  MoveL 674 to (56.44, 271.47, 190) mm, rotated rx -180 ry 0 rz -78.51 deg; joints [53.74, -26.691, 117.686, 53.744, 89.412, 89.198, -1451.486]
  MoveL 675 to (54.33, 277.32, 200) mm, rotated rx -180 ry 0 rz -72.32 deg; joints [53.369, -26.663, 117.257, 53.371, 89.646, 89.524, -1457.679]
  MoveL 676 to (51.74, 282.68, 210) mm, rotated rx 180 ry 0 rz -66.33 deg; joints [53.002, -26.629, 116.82, 53.002, 89.885, 89.848, -1463.668]
  MoveL 677 to (48.8, 287.5, 220) mm, rotated rx -180 ry 0 rz -60.59 deg; joints [52.638, -26.588, 116.376, 52.638, 90.129, 90.169, -1469.406]
  MoveL 678 to (45.62, 291.76, 230) mm, rotated rx -180 ry 0 rz -55.15 deg; joints [52.278, -26.54, 115.924, 52.28, 90.377, 90.487, -1474.846]
  MoveL 679 to (42.34, 295.45, 240) mm, rotated rx -180 ry 0 rz -50.06 deg; joints [51.921, -26.485, 115.464, 51.926, 90.63, 90.804, -1479.941]
  MoveL 680 to (39.07, 298.58, 250) mm, rotated rx -180 ry 0 rz -45.36 deg; joints [51.568, -26.422, 114.996, 51.577, 90.886, 91.117, -1484.643]
  MoveL 681 to (35.92, 301.18, 260) mm, rotated rx -180 ry 0 rz -41.09 deg; joints [51.218, -26.352, 114.52, 51.232, 91.147, 91.428, -1488.905]
  MoveL 682 to (33, 303.28, 270) mm, rotated rx -180 ry 0 rz -37.32 deg; joints [50.872, -26.275, 114.036, 50.893, 91.413, 91.737, -1492.679]
  MoveL 683 to (30.4, 304.94, 280) mm, rotated rx -180 ry 0 rz -34.08 deg; joints [50.529, -26.192, 113.545, 50.559, 91.682, 92.044, -1495.919]
  MoveL 684 to (28.22, 306.19, 290) mm, rotated rx -180 ry 0 rz -31.42 deg; joints [50.189, -26.102, 113.046, 50.229, 91.956, 92.348, -1498.582]
  MoveL 685 to (-21.11, 309.47, 290) mm, rotated rx 180 ry 0 rz 23.11 deg; joints [50.189, -26.125, 113.059, 50.229, 91.963, 92.356, -1553.11]
  Set speed (60.0 mm/s)
  MoveL 686 to (-18.74, 310.33, 280) mm, rotated rx -180 ry 0 rz 20.42 deg; joints [50.529, -26.229, 113.565, 50.559, 91.693, 92.057, -1550.424]
  MoveL 687 to (-15.8, 311.23, 270) mm, rotated rx -180 ry 0 rz 17.14 deg; joints [50.872, -26.331, 114.066, 50.894, 91.429, 91.757, -1547.138]
  MoveL 688 to (-12.3, 312.09, 260) mm, rotated rx 180 ry 0 rz 13.29 deg; joints [51.218, -26.429, 114.561, 51.233, 91.17, 91.456, -1543.29]
  MoveL 689 to (-8.28, 312.8, 250) mm, rotated rx -180 ry 0 rz 8.92 deg; joints [51.568, -26.522, 115.049, 51.577, 90.915, 91.154, -1538.917]
  MoveL 690 to (-3.78, 313.26, 240) mm, rotated rx -180 ry 0 rz 4.06 deg; joints [51.921, -26.61, 115.531, 51.926, 90.666, 90.85, -1534.059]
  MoveL 691 to (1.16, 313.37, 230) mm, rotated rx -180 ry 0 rz -1.24 deg; joints [52.278, -26.692, 116.005, 52.28, 90.42, 90.543, -1528.756]
  MoveL 692 to (6.46, 313.03, 220) mm, rotated rx -180 ry 0 rz -6.95 deg; joints [52.638, -26.768, 116.472, 52.639, 90.18, 90.235, -1523.053]
  MoveL 693 to (12.04, 312.14, 210) mm, rotated rx -180 ry 0 rz -13.01 deg; joints [53.002, -26.836, 116.931, 53.002, 89.943, 89.925, -1516.995]
  MoveL 694 to (17.8, 310.63, 200) mm, rotated rx -180 ry 0 rz -19.37 deg; joints [53.369, -26.897, 117.381, 53.37, 89.711, 89.611, -1510.629]
  MoveL 695 to (23.62, 308.44, 190) mm, rotated rx -180 ry 0 rz -25.99 deg; joints [53.74, -26.949, 117.823, 53.743, 89.483, 89.295, -1504.006]
  MoveL 696 to (29.38, 305.54, 180) mm, rotated rx -180 ry 0 rz -32.82 deg; joints [54.114, -26.993, 118.257, 54.121, 89.259, 88.976, -1497.176]
  MoveL 697 to (34.94, 301.92, 170) mm, rotated rx 180 ry 0 rz -39.81 deg; joints [54.492, -27.029, 118.682, 54.503, 89.04, 88.654, -1490.188]
  MoveL 698 to (40.17, 297.58, 160) mm, rotated rx -180 ry 0 rz -46.91 deg; joints [54.874, -27.057, 119.098, 54.891, 88.825, 88.33, -1483.094]
  MoveL 699 to (44.94, 292.58, 150) mm, rotated rx -180 ry 0 rz -54.06 deg; joints [55.259, -27.076, 119.507, 55.283, 88.615, 88.003, -1475.941]
  MoveL 700 to (49.15, 286.99, 140) mm, rotated rx -180 ry 0 rz -61.23 deg; joints [55.647, -27.089, 119.907, 55.68, 88.41, 87.673, -1468.774]
  MoveL 701 to (52.68, 280.9, 130) mm, rotated rx -180 ry 0 rz -68.36 deg; joints [56.04, -27.095, 120.299, 56.081, 88.211, 87.342, -1461.638]
  MoveL 702 to (55.46, 274.42, 120) mm, rotated rx -180 ry 0 rz -75.43 deg; joints [56.436, -27.096, 120.685, 56.488, 88.017, 87.009, -1454.572]
  MoveL 703 to (57.44, 267.68, 110) mm, rotated rx -180 ry 0 rz -82.39 deg; joints [56.835, -27.093, 121.064, 56.898, 87.829, 86.674, -1447.613]
  MoveL 704 to (58.6, 260.81, 100) mm, rotated rx 180 ry 0 rz -89.21 deg; joints [57.239, -27.086, 121.436, 57.314, 87.647, 86.34, -1440.794]
  MoveL 705 to (58.95, 253.96, 90) mm, rotated rx -180 ry 0 rz -95.85 deg; joints [57.646, -27.076, 121.803, 57.734, 87.472, 86.004, -1434.147]
  MoveL 706 to (58.51, 247.24, 80) mm, rotated rx -180 ry 0 rz -102.3 deg; joints [58.056, -27.066, 122.165, 58.158, 87.304, 85.669, -1427.701]
  MoveL 707 to (57.35, 240.79, 70) mm, rotated rx 180 ry 0 rz -108.52 deg; joints [58.471, -27.054, 122.522, 58.587, 87.144, 85.335, -1421.482]
  MoveL 708 to (55.55, 234.7, 60) mm, rotated rx -180 ry 0 rz -114.48 deg; joints [58.889, -27.042, 122.874, 59.02, 86.99, 85.002, -1415.517]
  MoveL 709 to (53.21, 229.07, 50) mm, rotated rx -180 ry 0 rz -120.17 deg; joints [59.311, -27.031, 123.223, 59.458, 86.844, 84.67, -1409.83]
  MoveL 710 to (50.45, 223.94, 40) mm, rotated rx -180 ry 0 rz -125.55 deg; joints [59.736, -27.021, 123.567, 59.899, 86.706, 84.34, -1404.447]
  MoveL 711 to (47.39, 219.37, 30) mm, rotated rx -180 ry 0 rz -130.61 deg; joints [60.166, -27.012, 123.907, 60.345, 86.576, 84.012, -1399.391]
  MoveL 712 to (44.15, 215.37, 20) mm, rotated rx -180 ry 0 rz -135.31 deg; joints [60.599, -27.005, 124.244, 60.794, 86.453, 83.685, -1394.688]
  MoveL 713 to (40.85, 211.93, 10) mm, rotated rx -180 ry 0 rz -139.64 deg; joints [61.035, -26.999, 124.577, 61.248, 86.339, 83.361, -1390.363]
  MoveL 714 to (37.62, 209.05, 0) mm, rotated rx -180 ry 0 rz -143.56 deg; joints [61.476, -26.994, 124.905, 61.705, 86.232, 83.039, -1386.442]
  MoveL 715 to (-21.11, 309.47, 290) mm, rotated rx 180 ry 0 rz 23.11 deg; joints [50.189, -26.125, 113.059, 50.229, 91.963, 92.356, -1553.11]
  Set speed (60.0 mm/s)
  MoveL 716 to (-34.79, 325.15, 290) mm, rotated rx -180 ry 0 rz 28.1 deg; joints [50.189, -24.773, 112.315, 50.215, 91.574, 91.889, -1558.101]
  MoveL 717 to (37.62, 209.05, 0) mm, rotated rx -180 ry 0 rz -143.56 deg; joints [61.476, -26.994, 124.905, 61.705, 86.232, 83.039, -1386.442]
  Set speed (60.0 mm/s)
  MoveL 718 to (55.59, 198.58, 0) mm, rotated rx -180 ry 0 rz -137.85 deg; joints [61.476, -25.55, 124.114, 61.745, 85.922, 82.463, -1392.15]
  MoveL 719 to (37.62, 209.05, 0) mm, rotated rx -180 ry 0 rz -143.56 deg; joints [61.476, -26.994, 124.905, 61.705, 86.232, 83.039, -1386.442]
  Set speed (60.0 mm/s)
  MoveL 720 to (40.85, 211.93, 10) mm, rotated rx 180 ry 0 rz -139.64 deg; joints [61.035, -26.999, 124.577, 61.248, 86.339, 83.361, -1390.363]
  MoveL 721 to (44.15, 215.37, 20) mm, rotated rx -180 ry 0 rz -135.31 deg; joints [60.599, -27.005, 124.244, 60.794, 86.453, 83.685, -1394.688]
  MoveL 722 to (47.39, 219.37, 30) mm, rotated rx -180 ry 0 rz -130.61 deg; joints [60.166, -27.012, 123.907, 60.345, 86.576, 84.012, -1399.391]
  MoveL 723 to (50.45, 223.94, 40) mm, rotated rx -180 ry 0 rz -125.55 deg; joints [59.736, -27.021, 123.567, 59.899, 86.706, 84.34, -1404.447]
  MoveL 724 to (53.21, 229.07, 50) mm, rotated rx -180 ry 0 rz -120.17 deg; joints [59.311, -27.031, 123.223, 59.458, 86.844, 84.67, -1409.83]
  MoveL 725 to (55.55, 234.7, 60) mm, rotated rx -180 ry 0 rz -114.48 deg; joints [58.889, -27.042, 122.874, 59.02, 86.99, 85.002, -1415.517]
  MoveL 726 to (57.35, 240.79, 70) mm, rotated rx -180 ry 0 rz -108.52 deg; joints [58.471, -27.054, 122.522, 58.587, 87.144, 85.335, -1421.482]
  MoveL 727 to (58.51, 247.24, 80) mm, rotated rx 180 ry 0 rz -102.3 deg; joints [58.056, -27.066, 122.165, 58.158, 87.304, 85.669, -1427.701]
  MoveL 728 to (58.95, 253.96, 90) mm, rotated rx -180 ry 0 rz -95.85 deg; joints [57.646, -27.076, 121.803, 57.734, 87.472, 86.004, -1434.147]
  MoveL 729 to (58.6, 260.81, 100) mm, rotated rx -180 ry 0 rz -89.21 deg; joints [57.239, -27.086, 121.436, 57.314, 87.647, 86.34, -1440.794]
  MoveL 730 to (57.44, 267.68, 110) mm, rotated rx -180 ry 0 rz -82.39 deg; joints [56.835, -27.093, 121.064, 56.898, 87.829, 86.674, -1447.613]
  MoveL 731 to (55.46, 274.42, 120) mm, rotated rx -180 ry 0 rz -75.43 deg; joints [56.436, -27.096, 120.685, 56.488, 88.017, 87.009, -1454.572]
  MoveL 732 to (52.68, 280.9, 130) mm, rotated rx -180 ry 0 rz -68.36 deg; joints [56.04, -27.095, 120.299, 56.081, 88.211, 87.342, -1461.638]
  MoveL 733 to (49.15, 286.99, 140) mm, rotated rx 180 ry 0 rz -61.23 deg; joints [55.647, -27.089, 119.907, 55.68, 88.41, 87.673, -1468.774]
  MoveL 734 to (44.94, 292.58, 150) mm, rotated rx -180 ry 0 rz -54.06 deg; joints [55.259, -27.076, 119.507, 55.283, 88.615, 88.003, -1475.941]
  MoveL 735 to (40.17, 297.58, 160) mm, rotated rx -180 ry 0 rz -46.91 deg; joints [54.874, -27.057, 119.098, 54.891, 88.825, 88.33, -1483.094]
  MoveL 736 to (34.94, 301.92, 170) mm, rotated rx -180 ry 0 rz -39.81 deg; joints [54.492, -27.029, 118.682, 54.503, 89.04, 88.654, -1490.188]
  MoveL 737 to (29.38, 305.54, 180) mm, rotated rx -180 ry 0 rz -32.82 deg; joints [54.114, -26.993, 118.257, 54.121, 89.259, 88.976, -1497.176]
  MoveL 738 to (23.62, 308.44, 190) mm, rotated rx -180 ry 0 rz -25.99 deg; joints [53.74, -26.949, 117.823, 53.743, 89.483, 89.295, -1504.006]
  MoveL 739 to (17.8, 310.63, 200) mm, rotated rx -180 ry 0 rz -19.37 deg; joints [53.369, -26.897, 117.381, 53.37, 89.711, 89.611, -1510.629]
  MoveL 740 to (12.04, 312.14, 210) mm, rotated rx 180 ry 0 rz -13.01 deg; joints [53.002, -26.836, 116.931, 53.002, 89.943, 89.925, -1516.995]
  MoveL 741 to (6.46, 313.03, 220) mm, rotated rx 180 ry 0 rz -6.95 deg; joints [52.638, -26.768, 116.472, 52.639, 90.18, 90.235, -1523.053]
  MoveL 742 to (1.16, 313.37, 230) mm, rotated rx 180 ry 0 rz -1.24 deg; joints [52.278, -26.692, 116.005, 52.28, 90.42, 90.543, -1528.756]
  MoveL 743 to (-3.78, 313.26, 240) mm, rotated rx -180 ry 0 rz 4.06 deg; joints [51.921, -26.61, 115.531, 51.926, 90.666, 90.85, -1534.059]
  MoveL 744 to (-8.28, 312.8, 250) mm, rotated rx -180 ry 0 rz 8.92 deg; joints [51.568, -26.522, 115.049, 51.577, 90.915, 91.154, -1538.917]
  MoveL 745 to (-12.3, 312.09, 260) mm, rotated rx -180 ry 0 rz 13.29 deg; joints [51.218, -26.429, 114.561, 51.233, 91.17, 91.456, -1543.29]
  MoveL 746 to (-15.8, 311.23, 270) mm, rotated rx -180 ry 0 rz 17.14 deg; joints [50.872, -26.331, 114.066, 50.894, 91.429, 91.757, -1547.138]
  MoveL 747 to (-18.74, 310.33, 280) mm, rotated rx -180 ry 0 rz 20.42 deg; joints [50.529, -26.229, 113.565, 50.559, 91.693, 92.057, -1550.424]
  MoveL 748 to (-21.11, 309.47, 290) mm, rotated rx -180 ry 0 rz 23.11 deg; joints [50.189, -26.125, 113.059, 50.229, 91.963, 92.356, -1553.11]
  MoveL 749 to (-34.79, 325.15, 290) mm, rotated rx -180 ry 0 rz 28.1 deg; joints [50.189, -24.773, 112.315, 50.215, 91.574, 91.889, -1558.101]
  Set speed (60.0 mm/s)
  MoveL 750 to (-31.73, 326.57, 280) mm, rotated rx -180 ry 0 rz 25.49 deg; joints [50.529, -24.874, 112.821, 50.547, 91.305, 91.585, -1555.486]
  MoveL 751 to (-27.92, 328.13, 270) mm, rotated rx -180 ry 0 rz 22.29 deg; joints [50.872, -24.972, 113.321, 50.883, 91.042, 91.281, -1552.288]
  MoveL 752 to (-23.38, 329.69, 260) mm, rotated rx 180 ry 0 rz 18.54 deg; joints [51.218, -25.067, 113.816, 51.225, 90.784, 90.976, -1548.542]
  MoveL 753 to (-18.11, 331.13, 250) mm, rotated rx -180 ry 0 rz 14.29 deg; joints [51.568, -25.158, 114.304, 51.571, 90.531, 90.669, -1544.286]
  MoveL 754 to (-12.17, 332.29, 240) mm, rotated rx -180 ry 0 rz 9.56 deg; joints [51.921, -25.244, 114.785, 51.922, 90.283, 90.361, -1539.557]
  MoveL 755 to (-5.61, 333.04, 230) mm, rotated rx 180 ry 0 rz 4.39 deg; joints [52.278, -25.324, 115.26, 52.278, 90.04, 90.051, -1534.392]
  MoveL 756 to (1.49, 333.22, 220) mm, rotated rx -180 ry 0 rz -1.17 deg; joints [52.638, -25.399, 115.727, 52.639, 89.801, 89.739, -1528.834]
  MoveL 757 to (9.03, 332.72, 210) mm, rotated rx -180 ry 0 rz -7.08 deg; joints [53.002, -25.466, 116.186, 53.004, 89.567, 89.425, -1522.922]
  MoveL 758 to (16.88, 331.41, 200) mm, rotated rx -180 ry 0 rz -13.3 deg; joints [53.369, -25.526, 116.636, 53.374, 89.337, 89.109, -1516.702]
  MoveL 759 to (24.89, 329.2, 190) mm, rotated rx -180 ry 0 rz -19.78 deg; joints [53.74, -25.578, 117.079, 53.749, 89.112, 88.789, -1510.217]
  MoveL 760 to (32.91, 326.04, 180) mm, rotated rx -180 ry 0 rz -26.49 deg; joints [54.114, -25.621, 117.512, 54.129, 88.892, 88.468, -1503.513]
  MoveL 761 to (40.75, 321.89, 170) mm, rotated rx -180 ry 0 rz -33.36 deg; joints [54.492, -25.656, 117.937, 54.514, 88.675, 88.143, -1496.637]
  MoveL 762 to (48.24, 316.75, 160) mm, rotated rx -180 ry 0 rz -40.37 deg; joints [54.874, -25.683, 118.353, 54.903, 88.464, 87.816, -1489.635]
  MoveL 763 to (55.2, 310.67, 150) mm, rotated rx -180 ry 0 rz -47.45 deg; joints [55.259, -25.702, 118.761, 55.297, 88.257, 87.486, -1482.551]
  MoveL 764 to (61.48, 303.74, 140) mm, rotated rx 180 ry 0 rz -54.57 deg; joints [55.647, -25.713, 119.16, 55.696, 88.056, 87.153, -1475.431]
  MoveL 765 to (66.92, 296.06, 130) mm, rotated rx -180 ry 0 rz -61.68 deg; joints [56.04, -25.718, 119.551, 56.099, 87.86, 86.819, -1468.317]
  MoveL 766 to (71.41, 287.77, 120) mm, rotated rx -180 ry 0 rz -68.75 deg; joints [56.436, -25.716, 119.935, 56.507, 87.669, 86.483, -1461.249]
  MoveL 767 to (74.87, 279.04, 110) mm, rotated rx -180 ry 0 rz -75.73 deg; joints [56.835, -25.71, 120.312, 56.92, 87.485, 86.145, -1454.266]
  MoveL 768 to (77.24, 270.04, 100) mm, rotated rx -180 ry 0 rz -82.6 deg; joints [57.239, -25.699, 120.682, 57.337, 87.306, 85.807, -1447.404]
  MoveL 769 to (78.53, 260.95, 90) mm, rotated rx -180 ry 0 rz -89.3 deg; joints [57.646, -25.686, 121.046, 57.759, 87.135, 85.468, -1440.696]
  MoveL 770 to (78.77, 251.96, 80) mm, rotated rx 180 ry 0 rz -95.83 deg; joints [58.056, -25.67, 121.404, 58.185, 86.97, 85.13, -1434.174]
  MoveL 771 to (78, 243.23, 70) mm, rotated rx -180 ry 0 rz -102.13 deg; joints [58.471, -25.653, 121.758, 58.616, 86.812, 84.791, -1427.868]
  MoveL 772 to (76.35, 234.91, 60) mm, rotated rx -180 ry 0 rz -108.19 deg; joints [58.889, -25.636, 122.106, 59.051, 86.662, 84.454, -1421.808]
  MoveL 773 to (73.92, 227.12, 50) mm, rotated rx -180 ry 0 rz -113.98 deg; joints [59.311, -25.619, 122.451, 59.49, 86.519, 84.117, -1416.021]
  MoveL 774 to (70.87, 219.96, 40) mm, rotated rx 180 ry 0 rz -119.46 deg; joints [59.736, -25.602, 122.791, 59.933, 86.384, 83.783, -1410.535]
  MoveL 775 to (67.34, 213.5, 30) mm, rotated rx -180 ry 0 rz -124.62 deg; joints [60.166, -25.587, 123.128, 60.38, 86.257, 83.45, -1405.378]
  MoveL 776 to (63.51, 207.78, 20) mm, rotated rx -180 ry 0 rz -129.42 deg; joints [60.599, -25.573, 123.46, 60.831, 86.137, 83.118, -1400.576]
  MoveL 777 to (59.54, 202.81, 10) mm, rotated rx -180 ry 0 rz -133.84 deg; joints [61.035, -25.561, 123.789, 61.286, 86.026, 82.79, -1396.157]
  MoveL 778 to (55.59, 198.58, 0) mm, rotated rx -180 ry 0 rz -137.85 deg; joints [61.476, -25.55, 124.114, 61.745, 85.922, 82.463, -1392.15]
  MoveL 779 to (-34.79, 325.15, 290) mm, rotated rx 180 ry 0 rz 28.1 deg; joints [50.189, -24.773, 112.315, 50.215, 91.574, 91.889, -1558.101]
  Set speed (60.0 mm/s)
  MoveL 780 to (-30.72, 304.75, 290) mm, rotated rx -180 ry 0 rz 34.47 deg; joints [50.189, -26.092, 113.041, 50.229, 91.953, 92.345, -1564.467]
  MoveL 781 to (55.59, 198.58, 0) mm, rotated rx -180 ry 0 rz -137.85 deg; joints [61.476, -25.55, 124.114, 61.745, 85.922, 82.463, -1392.15]
  Set speed (60.0 mm/s)
  MoveL 782 to (45.21, 216.6, 0) mm, rotated rx 180 ry 0 rz -133.83 deg; joints [61.476, -27.044, 124.932, 61.704, 86.242, 83.059, -1396.169]
  MoveL 783 to (55.59, 198.58, 0) mm, rotated rx -180 ry 0 rz -137.85 deg; joints [61.476, -25.55, 124.114, 61.745, 85.922, 82.463, -1392.15]
  Set speed (60.0 mm/s)
  MoveL 784 to (59.54, 202.81, 10) mm, rotated rx -180 ry 0 rz -133.84 deg; joints [61.035, -25.561, 123.789, 61.286, 86.026, 82.79, -1396.157]
  MoveL 785 to (63.51, 207.78, 20) mm, rotated rx -180 ry 0 rz -129.42 deg; joints [60.599, -25.573, 123.46, 60.831, 86.137, 83.118, -1400.576]
  MoveL 786 to (67.34, 213.5, 30) mm, rotated rx -180 ry 0 rz -124.62 deg; joints [60.166, -25.587, 123.128, 60.38, 86.257, 83.45, -1405.378]
  MoveL 787 to (70.87, 219.96, 40) mm, rotated rx -180 ry 0 rz -119.46 deg; joints [59.736, -25.602, 122.791, 59.933, 86.384, 83.783, -1410.535]
  MoveL 788 to (73.92, 227.12, 50) mm, rotated rx -180 ry 0 rz -113.98 deg; joints [59.311, -25.619, 122.451, 59.49, 86.519, 84.117, -1416.021]
  MoveL 789 to (76.35, 234.91, 60) mm, rotated rx -180 ry 0 rz -108.19 deg; joints [58.889, -25.636, 122.106, 59.051, 86.662, 84.454, -1421.808]
  MoveL 790 to (78, 243.23, 70) mm, rotated rx -180 ry 0 rz -102.13 deg; joints [58.471, -25.653, 121.758, 58.616, 86.812, 84.791, -1427.868]
  MoveL 791 to (78.77, 251.96, 80) mm, rotated rx -180 ry 0 rz -95.83 deg; joints [58.056, -25.67, 121.404, 58.185, 86.97, 85.13, -1434.174]
  MoveL 792 to (78.53, 260.95, 90) mm, rotated rx -180 ry 0 rz -89.3 deg; joints [57.646, -25.686, 121.046, 57.759, 87.135, 85.468, -1440.696]
  MoveL 793 to (77.24, 270.04, 100) mm, rotated rx 180 ry 0 rz -82.6 deg; joints [57.239, -25.699, 120.682, 57.337, 87.306, 85.807, -1447.404]
  MoveL 794 to (74.87, 279.04, 110) mm, rotated rx -180 ry 0 rz -75.73 deg; joints [56.835, -25.71, 120.312, 56.92, 87.485, 86.145, -1454.266]
  MoveL 795 to (71.41, 287.77, 120) mm, rotated rx 180 ry 0 rz -68.75 deg; joints [56.436, -25.716, 119.935, 56.507, 87.669, 86.483, -1461.249]
  MoveL 796 to (66.92, 296.06, 130) mm, rotated rx -180 ry 0 rz -61.68 deg; joints [56.04, -25.718, 119.551, 56.099, 87.86, 86.819, -1468.317]
  MoveL 797 to (61.48, 303.74, 140) mm, rotated rx 180 ry 0 rz -54.57 deg; joints [55.647, -25.713, 119.16, 55.696, 88.056, 87.153, -1475.431]
  MoveL 798 to (55.2, 310.67, 150) mm, rotated rx -180 ry 0 rz -47.45 deg; joints [55.259, -25.702, 118.761, 55.297, 88.257, 87.486, -1482.551]
  MoveL 799 to (48.24, 316.75, 160) mm, rotated rx -180 ry 0 rz -40.37 deg; joints [54.874, -25.683, 118.353, 54.903, 88.464, 87.816, -1489.635]
  MoveL 800 to (40.75, 321.89, 170) mm, rotated rx -180 ry 0 rz -33.36 deg; joints [54.492, -25.656, 117.937, 54.514, 88.675, 88.143, -1496.637]
  MoveL 801 to (32.91, 326.04, 180) mm, rotated rx -180 ry 0 rz -26.49 deg; joints [54.114, -25.621, 117.512, 54.129, 88.892, 88.468, -1503.513]
  MoveL 802 to (24.89, 329.2, 190) mm, rotated rx -180 ry 0 rz -19.78 deg; joints [53.74, -25.578, 117.079, 53.749, 89.112, 88.789, -1510.217]
  MoveL 803 to (16.88, 331.41, 200) mm, rotated rx -180 ry 0 rz -13.3 deg; joints [53.369, -25.526, 116.636, 53.374, 89.337, 89.109, -1516.702]
  MoveL 804 to (9.03, 332.72, 210) mm, rotated rx -180 ry 0 rz -7.08 deg; joints [53.002, -25.466, 116.186, 53.004, 89.567, 89.425, -1522.922]
  MoveL 805 to (1.49, 333.22, 220) mm, rotated rx -180 ry 0 rz -1.17 deg; joints [52.638, -25.399, 115.727, 52.639, 89.801, 89.739, -1528.834]
  MoveL 806 to (-5.61, 333.04, 230) mm, rotated rx 180 ry 0 rz 4.39 deg; joints [52.278, -25.324, 115.26, 52.278, 90.04, 90.051, -1534.392]
  MoveL 807 to (-12.17, 332.29, 240) mm, rotated rx 180 ry 0 rz 9.56 deg; joints [51.921, -25.244, 114.785, 51.922, 90.283, 90.361, -1539.557]
  MoveL 808 to (-18.11, 331.13, 250) mm, rotated rx -180 ry 0 rz 14.29 deg; joints [51.568, -25.158, 114.304, 51.571, 90.531, 90.669, -1544.286]
  MoveL 809 to (-23.38, 329.69, 260) mm, rotated rx -180 ry 0 rz 18.54 deg; joints [51.218, -25.067, 113.816, 51.225, 90.784, 90.976, -1548.542]
  MoveL 810 to (-27.92, 328.13, 270) mm, rotated rx -180 ry 0 rz 22.29 deg; joints [50.872, -24.972, 113.321, 50.883, 91.042, 91.281, -1552.288]
  MoveL 811 to (-31.73, 326.57, 280) mm, rotated rx -180 ry 0 rz 25.49 deg; joints [50.529, -24.874, 112.821, 50.547, 91.305, 91.585, -1555.486]
  MoveL 812 to (-34.79, 325.15, 290) mm, rotated rx -180 ry 0 rz 28.1 deg; joints [50.189, -24.773, 112.315, 50.215, 91.574, 91.889, -1558.101]
  MoveL 813 to (-30.72, 304.75, 290) mm, rotated rx 180 ry 0 rz 34.47 deg; joints [50.189, -26.092, 113.041, 50.229, 91.953, 92.345, -1564.467]
  Set speed (60.0 mm/s)
  MoveL 814 to (-28.54, 306.02, 280) mm, rotated rx -180 ry 0 rz 31.81 deg; joints [50.529, -26.199, 113.549, 50.559, 91.684, 92.046, -1561.806]
  MoveL 815 to (-25.81, 307.44, 270) mm, rotated rx 180 ry 0 rz 28.55 deg; joints [50.872, -26.304, 114.052, 50.893, 91.421, 91.748, -1558.548]
  MoveL 816 to (-22.53, 308.91, 260) mm, rotated rx -180 ry 0 rz 24.73 deg; joints [51.218, -26.406, 114.549, 51.233, 91.163, 91.448, -1554.728]
  MoveL 817 to (-18.7, 310.34, 250) mm, rotated rx -180 ry 0 rz 20.38 deg; joints [51.568, -26.504, 115.04, 51.577, 90.91, 91.147, -1550.381]
  MoveL 818 to (-14.35, 311.61, 240) mm, rotated rx 180 ry 0 rz 15.54 deg; joints [51.921, -26.598, 115.525, 51.926, 90.662, 90.845, -1545.543]
  MoveL 819 to (-9.52, 312.61, 230) mm, rotated rx -180 ry 0 rz 10.25 deg; joints [52.278, -26.687, 116.002, 52.28, 90.419, 90.541, -1540.254]
  MoveL 820 to (-4.24, 313.23, 220) mm, rotated rx -180 ry 0 rz 4.55 deg; joints [52.638, -26.769, 116.473, 52.639, 90.18, 90.236, -1534.554]
  MoveL 821 to (1.41, 313.37, 210) mm, rotated rx -180 ry 0 rz -1.51 deg; joints [53.002, -26.845, 116.935, 53.002, 89.946, 89.928, -1528.487]
  MoveL 822 to (7.35, 312.92, 200) mm, rotated rx -180 ry 0 rz -7.9 deg; joints [53.369, -26.913, 117.39, 53.37, 89.716, 89.617, -1522.098]
  MoveL 823 to (13.47, 311.83, 190) mm, rotated rx -180 ry 0 rz -14.57 deg; joints [53.74, -26.974, 117.836, 53.743, 89.49, 89.304, -1515.435]
  MoveL 824 to (19.65, 310.01, 180) mm, rotated rx -180 ry 0 rz -21.45 deg; joints [54.114, -27.026, 118.274, 54.121, 89.268, 88.988, -1508.548]
  MoveL 825 to (25.78, 307.45, 170) mm, rotated rx -180 ry 0 rz -28.51 deg; joints [54.492, -27.069, 118.703, 54.503, 89.051, 88.67, -1501.489]
  MoveL 826 to (31.7, 304.13, 160) mm, rotated rx 180 ry 0 rz -35.69 deg; joints [54.874, -27.104, 119.123, 54.89, 88.838, 88.348, -1494.307]
  MoveL 827 to (37.3, 300.08, 150) mm, rotated rx -180 ry 0 rz -42.95 deg; joints [55.259, -27.13, 119.535, 55.282, 88.63, 88.023, -1487.054]
  MoveL 828 to (42.45, 295.34, 140) mm, rotated rx -180 ry 0 rz -50.22 deg; joints [55.647, -27.148, 119.938, 55.679, 88.426, 87.696, -1479.778]
  MoveL 829 to (47.02, 289.99, 130) mm, rotated rx -180 ry 0 rz -57.48 deg; joints [56.04, -27.16, 120.334, 56.08, 88.228, 87.367, -1472.524]
  MoveL 830 to (50.93, 284.12, 120) mm, rotated rx -180 ry 0 rz -64.66 deg; joints [56.436, -27.164, 120.721, 56.487, 88.034, 87.035, -1465.337]
  MoveL 831 to (54.1, 277.85, 110) mm, rotated rx -180 ry 0 rz -71.74 deg; joints [56.835, -27.164, 121.101, 56.897, 87.847, 86.702, -1458.256]
  MoveL 832 to (56.49, 271.3, 100) mm, rotated rx -180 ry 0 rz -78.68 deg; joints [57.239, -27.158, 121.475, 57.313, 87.666, 86.368, -1451.316]
  MoveL 833 to (58.06, 264.62, 90) mm, rotated rx -180 ry 0 rz -85.45 deg; joints [57.646, -27.15, 121.842, 57.733, 87.491, 86.033, -1444.553]
  MoveL 834 to (58.85, 257.94, 80) mm, rotated rx -180 ry 0 rz -92 deg; joints [58.056, -27.138, 122.204, 58.157, 87.322, 85.698, -1437.997]
  MoveL 835 to (58.87, 251.39, 70) mm, rotated rx -180 ry 0 rz -98.32 deg; joints [58.471, -27.125, 122.56, 58.586, 87.161, 85.364, -1431.675]
  MoveL 836 to (58.2, 245.07, 60) mm, rotated rx -180 ry 0 rz -104.38 deg; joints [58.889, -27.112, 122.912, 59.019, 87.007, 85.03, -1425.616]
  MoveL 837 to (56.92, 239.11, 50) mm, rotated rx -180 ry 0 rz -110.16 deg; joints [59.311, -27.098, 123.259, 59.456, 86.86, 84.697, -1419.845]
  MoveL 838 to (55.13, 233.57, 40) mm, rotated rx -180 ry 0 rz -115.61 deg; joints [59.736, -27.085, 123.601, 59.898, 86.721, 84.366, -1414.385]
  MoveL 839 to (52.95, 228.52, 30) mm, rotated rx 180 ry 0 rz -120.74 deg; joints [60.166, -27.073, 123.94, 60.343, 86.59, 84.036, -1409.263]
  MoveL 840 to (50.48, 223.99, 20) mm, rotated rx -180 ry 0 rz -125.5 deg; joints [60.599, -27.062, 124.274, 60.793, 86.466, 83.708, -1404.503]
  MoveL 841 to (47.86, 220.02, 10) mm, rotated rx 180 ry 0 rz -129.87 deg; joints [61.035, -27.052, 124.605, 61.247, 86.35, 83.383, -1400.13]
  MoveL 842 to (45.21, 216.6, 0) mm, rotated rx 180 ry 0 rz -133.83 deg; joints [61.476, -27.044, 124.932, 61.704, 86.242, 83.059, -1396.169]
  MoveL 843 to (-30.72, 304.75, 290) mm, rotated rx -180 ry 0 rz 34.47 deg; joints [50.189, -26.092, 113.041, 50.229, 91.953, 92.345, -1564.467]
  Set speed (60.0 mm/s)
  MoveL 844 to (-58.22, 263.67, 290) mm, rotated rx -180 ry 0 rz 86.39 deg; joints [50.189, -25.818, 112.893, 50.226, 91.873, 92.248, -1616.394]
  MoveL 845 to (45.21, 216.6, 0) mm, rotated rx -180 ry 0 rz -133.83 deg; joints [61.476, -27.044, 124.932, 61.704, 86.242, 83.059, -1756.169]
  Set speed (60.0 mm/s)
  MoveL 846 to (58.12, 264.32, 0) mm, rotated rx 180 ry 0 rz -85.75 deg; joints [61.476, -27.37, 125.106, 61.695, 86.315, 83.194, -1804.254]
  MoveL 847 to (45.21, 216.6, 0) mm, rotated rx -180 ry 0 rz -133.83 deg; joints [61.476, -27.044, 124.932, 61.704, 86.242, 83.059, -1756.169]
  Set speed (60.0 mm/s)
  MoveL 848 to (47.86, 220.02, 10) mm, rotated rx -180 ry 0 rz -129.87 deg; joints [61.035, -27.052, 124.605, 61.247, 86.35, 83.383, -1760.13]
  MoveL 849 to (50.48, 223.99, 20) mm, rotated rx -180 ry 0 rz -125.5 deg; joints [60.599, -27.062, 124.274, 60.793, 86.466, 83.708, -1764.503]
  MoveL 850 to (52.95, 228.52, 30) mm, rotated rx -180 ry 0 rz -120.74 deg; joints [60.166, -27.073, 123.94, 60.343, 86.59, 84.036, -1769.263]
  MoveL 851 to (55.13, 233.57, 40) mm, rotated rx 180 ry 0 rz -115.61 deg; joints [59.736, -27.085, 123.601, 59.898, 86.721, 84.366, -1774.385]
  MoveL 852 to (56.92, 239.11, 50) mm, rotated rx -180 ry 0 rz -110.16 deg; joints [59.311, -27.098, 123.259, 59.456, 86.86, 84.697, -1779.845]
  MoveL 853 to (58.2, 245.07, 60) mm, rotated rx -180 ry 0 rz -104.38 deg; joints [58.889, -27.112, 122.912, 59.019, 87.007, 85.03, -1785.616]
  MoveL 854 to (58.87, 251.39, 70) mm, rotated rx -180 ry 0 rz -98.32 deg; joints [58.471, -27.125, 122.56, 58.586, 87.161, 85.364, -1791.675]
  MoveL 855 to (58.85, 257.94, 80) mm, rotated rx 180 ry 0 rz -92 deg; joints [58.056, -27.138, 122.204, 58.157, 87.322, 85.698, -1797.997]
  MoveL 856 to (58.06, 264.62, 90) mm, rotated rx -180 ry 0 rz -85.45 deg; joints [57.646, -27.15, 121.842, 57.733, 87.491, 86.033, -1804.553]
  MoveL 857 to (56.49, 271.3, 100) mm, rotated rx -180 ry 0 rz -78.68 deg; joints [57.239, -27.158, 121.475, 57.313, 87.666, 86.368, -1811.316]
  MoveL 858 to (54.1, 277.85, 110) mm, rotated rx -180 ry 0 rz -71.74 deg; joints [56.835, -27.164, 121.101, 56.897, 87.847, 86.702, -1818.256]
  MoveL 859 to (50.93, 284.12, 120) mm, rotated rx -180 ry 0 rz -64.66 deg; joints [56.436, -27.164, 120.721, 56.487, 88.034, 87.035, -1825.337]
  MoveL 860 to (47.02, 289.99, 130) mm, rotated rx 180 ry 0 rz -57.48 deg; joints [56.04, -27.16, 120.334, 56.08, 88.228, 87.367, -1832.524]
  MoveL 861 to (42.45, 295.34, 140) mm, rotated rx -180 ry 0 rz -50.22 deg; joints [55.647, -27.148, 119.938, 55.679, 88.426, 87.696, -1839.778]
  MoveL 862 to (37.3, 300.08, 150) mm, rotated rx -180 ry 0 rz -42.95 deg; joints [55.259, -27.13, 119.535, 55.282, 88.63, 88.023, -1847.054]
  MoveL 863 to (31.7, 304.13, 160) mm, rotated rx -180 ry 0 rz -35.69 deg; joints [54.874, -27.104, 119.123, 54.89, 88.838, 88.348, -1854.307]
  MoveL 864 to (25.78, 307.45, 170) mm, rotated rx -180 ry 0 rz -28.51 deg; joints [54.492, -27.069, 118.703, 54.503, 89.051, 88.67, -1861.489]
  MoveL 865 to (19.65, 310.01, 180) mm, rotated rx 180 ry 0 rz -21.45 deg; joints [54.114, -27.026, 118.274, 54.121, 89.268, 88.988, -1868.548]
  MoveL 866 to (13.47, 311.83, 190) mm, rotated rx -180 ry 0 rz -14.57 deg; joints [53.74, -26.974, 117.836, 53.743, 89.49, 89.304, -1875.435]
  MoveL 867 to (7.35, 312.92, 200) mm, rotated rx -180 ry 0 rz -7.9 deg; joints [53.369, -26.913, 117.39, 53.37, 89.716, 89.617, -1882.098]
  MoveL 868 to (1.41, 313.37, 210) mm, rotated rx -180 ry 0 rz -1.51 deg; joints [53.002, -26.845, 116.935, 53.002, 89.946, 89.928, -1888.487]
  MoveL 869 to (-4.24, 313.23, 220) mm, rotated rx 180 ry 0 rz 4.55 deg; joints [52.638, -26.769, 116.473, 52.639, 90.18, 90.236, -1894.554]
  MoveL 870 to (-9.52, 312.61, 230) mm, rotated rx 180 ry 0 rz 10.25 deg; joints [52.278, -26.687, 116.002, 52.28, 90.419, 90.541, -1900.254]
  MoveL 871 to (-14.35, 311.61, 240) mm, rotated rx -180 ry 0 rz 15.54 deg; joints [51.921, -26.598, 115.525, 51.926, 90.662, 90.845, -1905.543]
  MoveL 872 to (-18.7, 310.34, 250) mm, rotated rx -180 ry 0 rz 20.38 deg; joints [51.568, -26.504, 115.04, 51.577, 90.91, 91.147, -1910.381]
  MoveL 873 to (-22.53, 308.91, 260) mm, rotated rx 180 ry 0 rz 24.73 deg; joints [51.218, -26.406, 114.549, 51.233, 91.163, 91.448, -1914.728]
  MoveL 874 to (-25.81, 307.44, 270) mm, rotated rx -180 ry 0 rz 28.55 deg; joints [50.872, -26.304, 114.052, 50.893, 91.421, 91.748, -1918.548]
  MoveL 875 to (-28.54, 306.02, 280) mm, rotated rx -180 ry 0 rz 31.81 deg; joints [50.529, -26.199, 113.549, 50.559, 91.684, 92.046, -1921.806]
  MoveL 876 to (-30.72, 304.75, 290) mm, rotated rx -180 ry 0 rz 34.47 deg; joints [50.189, -26.092, 113.041, 50.229, 91.953, 92.345, -1924.467]
  MoveL 877 to (-58.22, 263.67, 290) mm, rotated rx -180 ry 0 rz 86.39 deg; joints [50.189, -25.818, 112.893, 50.226, 91.873, 92.248, -1976.394]
  Set speed (60.0 mm/s)
  MoveL 878 to (-57.77, 266.15, 280) mm, rotated rx 180 ry 0 rz 83.92 deg; joints [50.529, -25.932, 113.405, 50.556, 91.606, 91.951, -1973.924]
  MoveL 879 to (-57.08, 269.15, 270) mm, rotated rx -180 ry 0 rz 80.89 deg; joints [50.872, -26.045, 113.912, 50.891, 91.346, 91.655, -1970.894]
  MoveL 880 to (-56.08, 272.6, 260) mm, rotated rx -180 ry 0 rz 77.33 deg; joints [51.218, -26.159, 114.416, 51.231, 91.092, 91.359, -1967.333]
  MoveL 881 to (-54.69, 276.44, 250) mm, rotated rx -180 ry 0 rz 73.27 deg; joints [51.568, -26.271, 114.915, 51.576, 90.843, 91.063, -1963.267]
  MoveL 882 to (-52.84, 280.57, 240) mm, rotated rx 180 ry 0 rz 68.72 deg; joints [51.921, -26.383, 115.409, 51.925, 90.601, 90.767, -1958.724]
  MoveL 883 to (-50.46, 284.91, 230) mm, rotated rx -180 ry 0 rz 63.73 deg; joints [52.278, -26.493, 115.899, 52.28, 90.364, 90.47, -1953.731]
  MoveL 884 to (-47.51, 289.33, 220) mm, rotated rx -180 ry 0 rz 58.32 deg; joints [52.638, -26.601, 116.383, 52.638, 90.132, 90.173, -1948.316]
  MoveL 885 to (-43.95, 293.72, 210) mm, rotated rx -180 ry 0 rz 52.51 deg; joints [53.002, -26.705, 116.861, 53.002, 89.906, 89.876, -1942.509]
  MoveL 886 to (-39.77, 297.95, 200) mm, rotated rx -180 ry 0 rz 46.34 deg; joints [53.369, -26.806, 117.333, 53.37, 89.686, 89.577, -1936.342]
  MoveL 887 to (-34.96, 301.9, 190) mm, rotated rx -180 ry 0 rz 39.85 deg; joints [53.74, -26.902, 117.798, 53.743, 89.47, 89.277, -1929.847]
  MoveL 888 to (-29.57, 305.43, 180) mm, rotated rx 180 ry 0 rz 33.06 deg; joints [54.114, -26.992, 118.256, 54.121, 89.259, 88.976, -1923.063]
  MoveL 889 to (-23.65, 308.43, 170) mm, rotated rx -180 ry 0 rz 26.03 deg; joints [54.492, -27.076, 118.707, 54.503, 89.053, 88.672, -1916.03]
  MoveL 890 to (-17.28, 310.79, 160) mm, rotated rx -180 ry 0 rz 18.79 deg; joints [54.874, -27.152, 119.149, 54.89, 88.851, 88.366, -1908.791]
  MoveL 891 to (-10.57, 312.43, 150) mm, rotated rx -180 ry 0 rz 11.39 deg; joints [55.259, -27.22, 119.583, 55.282, 88.654, 88.058, -1901.395]
  MoveL 892 to (-3.62, 313.27, 140) mm, rotated rx -180 ry 0 rz 3.89 deg; joints [55.647, -27.279, 120.008, 55.678, 88.461, 87.747, -1893.889]
  MoveL 893 to (3.42, 313.28, 130) mm, rotated rx -180 ry 0 rz -3.67 deg; joints [56.04, -27.329, 120.423, 56.078, 88.272, 87.433, -1886.327]
  MoveL 894 to (10.42, 312.46, 120) mm, rotated rx -180 ry 0 rz -11.24 deg; joints [56.436, -27.37, 120.83, 56.484, 88.088, 87.116, -1878.761]
  MoveL 895 to (17.25, 310.8, 110) mm, rotated rx -180 ry 0 rz -18.76 deg; joints [56.835, -27.402, 121.227, 56.894, 87.908, 86.796, -1871.243]
  MoveL 896 to (23.78, 308.38, 100) mm, rotated rx -180 ry 0 rz -26.18 deg; joints [57.239, -27.425, 121.616, 57.308, 87.733, 86.474, -1863.825]
  MoveL 897 to (29.89, 305.25, 90) mm, rotated rx -180 ry 0 rz -33.45 deg; joints [57.646, -27.44, 121.996, 57.728, 87.564, 86.149, -1856.554]
  MoveL 898 to (35.48, 301.51, 80) mm, rotated rx -180 ry 0 rz -40.52 deg; joints [58.056, -27.448, 122.368, 58.151, 87.399, 85.822, -1849.477]
  MoveL 899 to (40.49, 297.28, 70) mm, rotated rx -180 ry 0 rz -47.36 deg; joints [58.471, -27.45, 122.732, 58.579, 87.241, 85.494, -1842.636]
  MoveL 900 to (44.86, 292.68, 60) mm, rotated rx -180 ry 0 rz -53.93 deg; joints [58.889, -27.447, 123.089, 59.012, 87.088, 85.165, -1836.069]
  MoveL 901 to (48.58, 287.83, 50) mm, rotated rx -180 ry 0 rz -60.19 deg; joints [59.311, -27.439, 123.44, 59.449, 86.941, 84.835, -1829.813]
  MoveL 902 to (51.63, 282.88, 40) mm, rotated rx -180 ry 0 rz -66.1 deg; joints [59.736, -27.428, 123.784, 59.89, 86.802, 84.505, -1823.9]
  MoveL 903 to (54.06, 277.94, 30) mm, rotated rx -180 ry 0 rz -71.64 deg; joints [60.166, -27.415, 124.122, 60.335, 86.669, 84.175, -1818.36]
  MoveL 904 to (55.91, 273.13, 20) mm, rotated rx -180 ry 0 rz -76.78 deg; joints [60.599, -27.4, 124.455, 60.785, 86.543, 83.847, -1813.221]
  MoveL 905 to (57.23, 268.56, 10) mm, rotated rx -180 ry 0 rz -81.49 deg; joints [61.035, -27.385, 124.783, 61.238, 86.425, 83.519, -1808.51]
  MoveL 906 to (58.12, 264.32, 0) mm, rotated rx -180 ry 0 rz -85.75 deg; joints [61.476, -27.37, 125.106, 61.695, 86.315, 83.194, -1804.254]
  MoveL 907 to (-58.22, 263.67, 290) mm, rotated rx -180 ry 0 rz 86.39 deg; joints [50.189, -25.818, 112.893, 50.226, 91.873, 92.248, -1976.394]
  Set speed (60.0 mm/s)
  MoveL 908 to (-78.63, 259.66, 290) mm, rotated rx 180 ry 0 rz 90.25 deg; joints [50.189, -24.451, 112.133, 50.212, 91.484, 91.781, -1980.245]
  MoveL 909 to (58.12, 264.32, 0) mm, rotated rx 180 ry 0 rz -85.75 deg; joints [61.476, -27.37, 125.106, 61.695, 86.315, 83.194, -1804.254]
  Set speed (60.0 mm/s)
  MoveL 910 to (76.17, 274.65, 0) mm, rotated rx 180 ry 0 rz -79.11 deg; joints [61.476, -25.94, 124.331, 61.734, 86.004, 82.616, -1810.889]
  MoveL 911 to (58.12, 264.32, 0) mm, rotated rx -180 ry 0 rz -85.75 deg; joints [61.476, -27.37, 125.106, 61.695, 86.315, 83.194, -1804.254]
  Set speed (60.0 mm/s)
  MoveL 912 to (57.23, 268.56, 10) mm, rotated rx -180 ry 0 rz -81.49 deg; joints [61.035, -27.385, 124.783, 61.238, 86.425, 83.519, -1808.51]
  MoveL 913 to (55.91, 273.13, 20) mm, rotated rx -180 ry 0 rz -76.78 deg; joints [60.599, -27.4, 124.455, 60.785, 86.543, 83.847, -1813.221]
  MoveL 914 to (54.06, 277.94, 30) mm, rotated rx -180 ry 0 rz -71.64 deg; joints [60.166, -27.415, 124.122, 60.335, 86.669, 84.175, -1818.36]
  MoveL 915 to (51.63, 282.88, 40) mm, rotated rx -180 ry 0 rz -66.1 deg; joints [59.736, -27.428, 123.784, 59.89, 86.802, 84.505, -1823.9]
  MoveL 916 to (48.58, 287.83, 50) mm, rotated rx 180 ry 0 rz -60.19 deg; joints [59.311, -27.439, 123.44, 59.449, 86.941, 84.835, -1829.813]
  MoveL 917 to (44.86, 292.68, 60) mm, rotated rx 180 ry 0 rz -53.93 deg; joints [58.889, -27.447, 123.089, 59.012, 87.088, 85.165, -1836.069]
  MoveL 918 to (40.49, 297.28, 70) mm, rotated rx -180 ry 0 rz -47.36 deg; joints [58.471, -27.45, 122.732, 58.579, 87.241, 85.494, -1842.636]
  MoveL 919 to (35.48, 301.51, 80) mm, rotated rx -180 ry 0 rz -40.52 deg; joints [58.056, -27.448, 122.368, 58.151, 87.399, 85.822, -1849.477]
  MoveL 920 to (29.89, 305.25, 90) mm, rotated rx -180 ry 0 rz -33.45 deg; joints [57.646, -27.44, 121.996, 57.728, 87.564, 86.149, -1856.554]
  MoveL 921 to (23.78, 308.38, 100) mm, rotated rx -180 ry 0 rz -26.18 deg; joints [57.239, -27.425, 121.616, 57.308, 87.733, 86.474, -1863.825]
  MoveL 922 to (17.25, 310.8, 110) mm, rotated rx -180 ry 0 rz -18.76 deg; joints [56.835, -27.402, 121.227, 56.894, 87.908, 86.796, -1871.243]
  MoveL 923 to (10.42, 312.46, 120) mm, rotated rx -180 ry 0 rz -11.24 deg; joints [56.436, -27.37, 120.83, 56.484, 88.088, 87.116, -1878.761]
  MoveL 924 to (3.42, 313.28, 130) mm, rotated rx -180 ry 0 rz -3.67 deg; joints [56.04, -27.329, 120.423, 56.078, 88.272, 87.433, -1886.327]
  MoveL 925 to (-3.62, 313.27, 140) mm, rotated rx -180 ry 0 rz 3.89 deg; joints [55.647, -27.279, 120.008, 55.678, 88.461, 87.747, -1893.889]
  MoveL 926 to (-10.57, 312.43, 150) mm, rotated rx -180 ry 0 rz 11.39 deg; joints [55.259, -27.22, 119.583, 55.282, 88.654, 88.058, -1901.395]
  MoveL 927 to (-17.28, 310.79, 160) mm, rotated rx -180 ry 0 rz 18.79 deg; joints [54.874, -27.152, 119.149, 54.89, 88.851, 88.366, -1908.791]
  MoveL 928 to (-23.65, 308.43, 170) mm, rotated rx -180 ry 0 rz 26.03 deg; joints [54.492, -27.076, 118.707, 54.503, 89.053, 88.672, -1916.03]
  MoveL 929 to (-29.57, 305.43, 180) mm, rotated rx -180 ry 0 rz 33.06 deg; joints [54.114, -26.992, 118.256, 54.121, 89.259, 88.976, -1923.063]
  MoveL 930 to (-34.96, 301.9, 190) mm, rotated rx 180 ry 0 rz 39.85 deg; joints [53.74, -26.902, 117.798, 53.743, 89.47, 89.277, -1929.847]
  MoveL 931 to (-39.77, 297.95, 200) mm, rotated rx -180 ry 0 rz 46.34 deg; joints [53.369, -26.806, 117.333, 53.37, 89.686, 89.577, -1936.342]
  MoveL 932 to (-43.95, 293.72, 210) mm, rotated rx -180 ry 0 rz 52.51 deg; joints [53.002, -26.705, 116.861, 53.002, 89.906, 89.876, -1942.509]
  MoveL 933 to (-47.51, 289.33, 220) mm, rotated rx -180 ry 0 rz 58.32 deg; joints [52.638, -26.601, 116.383, 52.638, 90.132, 90.173, -1948.316]
  MoveL 934 to (-50.46, 284.91, 230) mm, rotated rx 180 ry 0 rz 63.73 deg; joints [52.278, -26.493, 115.899, 52.28, 90.364, 90.47, -1953.731]
  MoveL 935 to (-52.84, 280.57, 240) mm, rotated rx -180 ry 0 rz 68.72 deg; joints [51.921, -26.383, 115.409, 51.925, 90.601, 90.767, -1958.724]
  MoveL 936 to (-54.69, 276.44, 250) mm, rotated rx -180 ry 0 rz 73.27 deg; joints [51.568, -26.271, 114.915, 51.576, 90.843, 91.063, -1963.267]
  MoveL 937 to (-56.08, 272.6, 260) mm, rotated rx -180 ry 0 rz 77.33 deg; joints [51.218, -26.159, 114.416, 51.231, 91.092, 91.359, -1967.333]
  MoveL 938 to (-57.08, 269.15, 270) mm, rotated rx -180 ry 0 rz 80.89 deg; joints [50.872, -26.045, 113.912, 50.891, 91.346, 91.655, -1970.894]
  MoveL 939 to (-57.77, 266.15, 280) mm, rotated rx -180 ry 0 rz 83.92 deg; joints [50.529, -25.932, 113.405, 50.556, 91.606, 91.951, -1973.924]
  MoveL 940 to (-58.22, 263.67, 290) mm, rotated rx -180 ry 0 rz 86.39 deg; joints [50.189, -25.818, 112.893, 50.226, 91.873, 92.248, -1976.394]
  MoveL 941 to (-78.63, 259.66, 290) mm, rotated rx -180 ry 0 rz 90.25 deg; joints [50.189, -24.451, 112.133, 50.212, 91.484, 91.781, -1980.245]
  Set speed (60.0 mm/s)
  MoveL 942 to (-78.34, 263.02, 280) mm, rotated rx -180 ry 0 rz 87.79 deg; joints [50.529, -24.56, 112.644, 50.544, 91.218, 91.479, -1977.792]
  MoveL 943 to (-77.78, 267.1, 270) mm, rotated rx 180 ry 0 rz 84.79 deg; joints [50.872, -24.669, 113.15, 50.881, 90.958, 91.178, -1974.787]
  MoveL 944 to (-76.86, 271.82, 260) mm, rotated rx -180 ry 0 rz 81.26 deg; joints [51.218, -24.777, 113.653, 51.224, 90.704, 90.877, -1971.259]
  MoveL 945 to (-75.48, 277.1, 250) mm, rotated rx 180 ry 0 rz 77.24 deg; joints [51.568, -24.886, 114.151, 51.57, 90.456, 90.575, -1967.238]
  MoveL 946 to (-73.51, 282.82, 240) mm, rotated rx -180 ry 0 rz 72.75 deg; joints [51.921, -24.993, 114.645, 51.922, 90.215, 90.274, -1962.753]
  MoveL 947 to (-70.88, 288.88, 230) mm, rotated rx 180 ry 0 rz 67.83 deg; joints [52.278, -25.099, 115.134, 52.278, 89.979, 89.972, -1957.833]
  MoveL 948 to (-67.49, 295.12, 220) mm, rotated rx 180 ry 0 rz 62.51 deg; joints [52.638, -25.203, 115.617, 52.639, 89.748, 89.67, -1952.509]
  MoveL 949 to (-63.28, 301.4, 210) mm, rotated rx -180 ry 0 rz 56.81 deg; joints [53.002, -25.304, 116.095, 53.005, 89.524, 89.368, -1946.81]
  MoveL 950 to (-58.22, 307.54, 200) mm, rotated rx -180 ry 0 rz 50.77 deg; joints [53.369, -25.401, 116.567, 53.375, 89.304, 89.064, -1940.77]
  MoveL 951 to (-52.31, 313.38, 190) mm, rotated rx -180 ry 0 rz 44.42 deg; joints [53.74, -25.495, 117.033, 53.75, 89.09, 88.76, -1934.421]
  MoveL 952 to (-45.56, 318.73, 180) mm, rotated rx -180 ry 0 rz 37.8 deg; joints [54.114, -25.583, 117.491, 54.129, 88.882, 88.454, -1927.8]
  MoveL 953 to (-38.04, 323.45, 170) mm, rotated rx -180 ry 0 rz 30.95 deg; joints [54.492, -25.664, 117.942, 54.514, 88.678, 88.146, -1920.945]
  MoveL 954 to (-29.85, 327.37, 160) mm, rotated rx 180 ry 0 rz 23.9 deg; joints [54.874, -25.739, 118.384, 54.902, 88.478, 87.836, -1913.897]
  MoveL 955 to (-21.11, 330.36, 150) mm, rotated rx -180 ry 0 rz 16.7 deg; joints [55.259, -25.806, 118.819, 55.296, 88.284, 87.524, -1906.697]
  MoveL 956 to (-11.96, 332.32, 140) mm, rotated rx -180 ry 0 rz 9.39 deg; joints [55.647, -25.865, 119.244, 55.694, 88.094, 87.209, -1899.391]
  MoveL 957 to (-2.59, 333.2, 130) mm, rotated rx -180 ry 0 rz 2.03 deg; joints [56.04, -25.915, 119.66, 56.096, 87.909, 86.892, -1892.026]
  MoveL 958 to (6.83, 332.94, 120) mm, rotated rx -180 ry 0 rz -5.35 deg; joints [56.436, -25.956, 120.067, 56.504, 87.728, 86.572, -1884.647]
  MoveL 959 to (16.13, 331.57, 110) mm, rotated rx -180 ry 0 rz -12.7 deg; joints [56.835, -25.988, 120.465, 56.916, 87.552, 86.25, -1877.302]
  MoveL 960 to (25.11, 329.13, 100) mm, rotated rx -180 ry 0 rz -19.96 deg; joints [57.239, -26.011, 120.854, 57.332, 87.381, 85.925, -1870.039]
  MoveL 961 to (33.62, 325.71, 90) mm, rotated rx -180 ry 0 rz -27.1 deg; joints [57.646, -26.026, 121.234, 57.753, 87.216, 85.597, -1862.902]
  MoveL 962 to (41.52, 321.41, 80) mm, rotated rx -180 ry 0 rz -34.06 deg; joints [58.056, -26.034, 121.606, 58.178, 87.056, 85.268, -1855.936]
  MoveL 963 to (48.7, 316.39, 70) mm, rotated rx -180 ry 0 rz -40.82 deg; joints [58.471, -26.035, 121.969, 58.608, 86.901, 84.937, -1849.182]
  MoveL 964 to (55.08, 310.79, 60) mm, rotated rx 180 ry 0 rz -47.32 deg; joints [58.889, -26.031, 122.326, 59.042, 86.752, 84.605, -1842.679]
  MoveL 965 to (60.61, 304.79, 50) mm, rotated rx -180 ry 0 rz -53.53 deg; joints [59.311, -26.022, 122.675, 59.48, 86.61, 84.272, -1836.465]
  MoveL 966 to (65.29, 298.57, 40) mm, rotated rx -180 ry 0 rz -59.43 deg; joints [59.736, -26.009, 123.017, 59.923, 86.475, 83.94, -1830.575]
  MoveL 967 to (69.12, 292.29, 30) mm, rotated rx -180 ry 0 rz -64.96 deg; joints [60.166, -25.994, 123.353, 60.37, 86.346, 83.607, -1825.041]
  MoveL 968 to (72.16, 286.11, 20) mm, rotated rx 180 ry 0 rz -70.1 deg; joints [60.599, -25.977, 123.684, 60.821, 86.225, 83.275, -1819.895]
  MoveL 969 to (74.48, 280.19, 10) mm, rotated rx -180 ry 0 rz -74.83 deg; joints [61.035, -25.958, 124.01, 61.275, 86.111, 82.945, -1815.168]
  MoveL 970 to (76.17, 274.65, 0) mm, rotated rx 180 ry 0 rz -79.11 deg; joints [61.476, -25.94, 124.331, 61.734, 86.004, 82.616, -1810.889]
  MoveL 971 to (-78.63, 259.66, 290) mm, rotated rx 180 ry 0 rz 90.25 deg; joints [50.189, -24.451, 112.133, 50.212, 91.484, 91.781, -1980.245]
  Set speed (60.0 mm/s)
  MoveL 972 to (-58.93, 252.99, 290) mm, rotated rx 180 ry 0 rz 96.78 deg; joints [50.189, -25.75, 112.856, 50.225, 91.853, 92.224, -1986.784]
  MoveL 973 to (76.17, 274.65, 0) mm, rotated rx 180 ry 0 rz -79.11 deg; joints [61.476, -25.94, 124.331, 61.734, 86.004, 82.616, -1810.889]
  Set speed (60.0 mm/s)
  MoveL 974 to (55.37, 274.67, 0) mm, rotated rx -180 ry 0 rz -75.16 deg; joints [61.476, -27.444, 125.145, 61.693, 86.331, 83.225, -1814.838]
  MoveL 975 to (76.17, 274.65, 0) mm, rotated rx -180 ry 0 rz -79.11 deg; joints [61.476, -25.94, 124.331, 61.734, 86.004, 82.616, -1810.889]
  Set speed (60.0 mm/s)
  MoveL 976 to (74.48, 280.19, 10) mm, rotated rx -180 ry 0 rz -74.83 deg; joints [61.035, -25.958, 124.01, 61.275, 86.111, 82.945, -1815.168]
  MoveL 977 to (72.16, 286.11, 20) mm, rotated rx -180 ry 0 rz -70.1 deg; joints [60.599, -25.977, 123.684, 60.821, 86.225, 83.275, -1819.895]
  MoveL 978 to (69.12, 292.29, 30) mm, rotated rx -180 ry 0 rz -64.96 deg; joints [60.166, -25.994, 123.353, 60.37, 86.346, 83.607, -1825.041]
  MoveL 979 to (65.29, 298.57, 40) mm, rotated rx -180 ry 0 rz -59.43 deg; joints [59.736, -26.009, 123.017, 59.923, 86.475, 83.94, -1830.575]
  MoveL 980 to (60.61, 304.79, 50) mm, rotated rx -180 ry 0 rz -53.53 deg; joints [59.311, -26.022, 122.675, 59.48, 86.61, 84.272, -1836.465]
  MoveL 981 to (55.08, 310.79, 60) mm, rotated rx -180 ry 0 rz -47.32 deg; joints [58.889, -26.031, 122.326, 59.042, 86.752, 84.605, -1842.679]
  MoveL 982 to (48.7, 316.39, 70) mm, rotated rx -180 ry 0 rz -40.82 deg; joints [58.471, -26.035, 121.969, 58.608, 86.901, 84.937, -1849.182]
  MoveL 983 to (41.52, 321.41, 80) mm, rotated rx -180 ry 0 rz -34.06 deg; joints [58.056, -26.034, 121.606, 58.178, 87.056, 85.268, -1855.936]
  MoveL 984 to (33.62, 325.71, 90) mm, rotated rx -180 ry 0 rz -27.1 deg; joints [57.646, -26.026, 121.234, 57.753, 87.216, 85.597, -1862.902]
  MoveL 985 to (25.11, 329.13, 100) mm, rotated rx -180 ry 0 rz -19.96 deg; joints [57.239, -26.011, 120.854, 57.332, 87.381, 85.925, -1870.039]
  MoveL 986 to (16.13, 331.57, 110) mm, rotated rx -180 ry 0 rz -12.7 deg; joints [56.835, -25.988, 120.465, 56.916, 87.552, 86.25, -1877.302]
  MoveL 987 to (6.83, 332.94, 120) mm, rotated rx 180 ry 0 rz -5.35 deg; joints [56.436, -25.956, 120.067, 56.504, 87.728, 86.572, -1884.647]
  MoveL 988 to (-2.59, 333.2, 130) mm, rotated rx 180 ry 0 rz 2.03 deg; joints [56.04, -25.915, 119.66, 56.096, 87.909, 86.892, -1892.026]
  MoveL 989 to (-11.96, 332.32, 140) mm, rotated rx -180 ry 0 rz 9.39 deg; joints [55.647, -25.865, 119.244, 55.694, 88.094, 87.209, -1899.391]
  MoveL 990 to (-21.11, 330.36, 150) mm, rotated rx -180 ry 0 rz 16.7 deg; joints [55.259, -25.806, 118.819, 55.296, 88.284, 87.524, -1906.697]
  MoveL 991 to (-29.85, 327.37, 160) mm, rotated rx -180 ry 0 rz 23.9 deg; joints [54.874, -25.739, 118.384, 54.902, 88.478, 87.836, -1913.897]
  MoveL 992 to (-38.04, 323.45, 170) mm, rotated rx -180 ry 0 rz 30.95 deg; joints [54.492, -25.664, 117.942, 54.514, 88.678, 88.146, -1920.945]
  MoveL 993 to (-45.56, 318.73, 180) mm, rotated rx 180 ry 0 rz 37.8 deg; joints [54.114, -25.583, 117.491, 54.129, 88.882, 88.454, -1927.8]
  MoveL 994 to (-52.31, 313.38, 190) mm, rotated rx -180 ry 0 rz 44.42 deg; joints [53.74, -25.495, 117.033, 53.75, 89.09, 88.76, -1934.421]
  MoveL 995 to (-58.22, 307.54, 200) mm, rotated rx 180 ry 0 rz 50.77 deg; joints [53.369, -25.401, 116.567, 53.375, 89.304, 89.064, -1940.77]
  MoveL 996 to (-63.28, 301.4, 210) mm, rotated rx -180 ry 0 rz 56.81 deg; joints [53.002, -25.304, 116.095, 53.005, 89.524, 89.368, -1946.81]
  MoveL 997 to (-67.49, 295.12, 220) mm, rotated rx 180 ry 0 rz 62.51 deg; joints [52.638, -25.203, 115.617, 52.639, 89.748, 89.67, -1952.509]
  MoveL 998 to (-70.88, 288.88, 230) mm, rotated rx -180 ry 0 rz 67.83 deg; joints [52.278, -25.099, 115.134, 52.278, 89.979, 89.972, -1957.833]
  MoveL 999 to (-73.51, 282.82, 240) mm, rotated rx -180 ry 0 rz 72.75 deg; joints [51.921, -24.993, 114.645, 51.922, 90.215, 90.274, -1962.753]
  MoveL 1000 to (-75.48, 277.1, 250) mm, rotated rx -180 ry 0 rz 77.24 deg; joints [51.568, -24.886, 114.151, 51.57, 90.456, 90.575, -1967.238]
  MoveL 1001 to (-76.86, 271.82, 260) mm, rotated rx -180 ry 0 rz 81.26 deg; joints [51.218, -24.777, 113.653, 51.224, 90.704, 90.877, -1971.259]
  MoveL 1002 to (-77.78, 267.1, 270) mm, rotated rx -180 ry 0 rz 84.79 deg; joints [50.872, -24.669, 113.15, 50.881, 90.958, 91.178, -1974.787]
  MoveL 1003 to (-78.34, 263.02, 280) mm, rotated rx 180 ry 0 rz 87.79 deg; joints [50.529, -24.56, 112.644, 50.544, 91.218, 91.479, -1977.792]
  MoveL 1004 to (-78.63, 259.66, 290) mm, rotated rx -180 ry 0 rz 90.25 deg; joints [50.189, -24.451, 112.133, 50.212, 91.484, 91.781, -1980.245]
  MoveL 1005 to (-58.93, 252.99, 290) mm, rotated rx -180 ry 0 rz 96.78 deg; joints [50.189, -25.75, 112.856, 50.225, 91.853, 92.224, -1986.784]
  Set speed (60.0 mm/s)
  MoveL 1006 to (-58.94, 255.51, 280) mm, rotated rx -180 ry 0 rz 94.36 deg; joints [50.529, -25.864, 113.367, 50.555, 91.586, 91.927, -1984.356]
  MoveL 1007 to (-58.8, 258.59, 270) mm, rotated rx -180 ry 0 rz 91.38 deg; joints [50.872, -25.977, 113.875, 50.891, 91.326, 91.631, -1981.378]
  MoveL 1008 to (-58.44, 262.16, 260) mm, rotated rx -180 ry 0 rz 87.88 deg; joints [51.218, -26.09, 114.379, 51.231, 91.072, 91.334, -1977.879]
  MoveL 1009 to (-57.77, 266.19, 250) mm, rotated rx -180 ry 0 rz 83.88 deg; joints [51.568, -26.204, 114.878, 51.575, 90.824, 91.038, -1973.884]
  MoveL 1010 to (-56.69, 270.59, 240) mm, rotated rx 180 ry 0 rz 79.42 deg; joints [51.921, -26.316, 115.373, 51.925, 90.582, 90.742, -1969.42]
  MoveL 1011 to (-55.14, 275.28, 230) mm, rotated rx -180 ry 0 rz 74.51 deg; joints [52.278, -26.428, 115.864, 52.279, 90.345, 90.446, -1964.512]
  MoveL 1012 to (-53.04, 280.16, 220) mm, rotated rx -180 ry 0 rz 69.19 deg; joints [52.638, -26.538, 116.349, 52.638, 90.115, 90.15, -1959.189]
  MoveL 1013 to (-50.33, 285.12, 210) mm, rotated rx -180 ry 0 rz 63.48 deg; joints [53.002, -26.646, 116.829, 53.002, 89.89, 89.854, -1953.477]
  MoveL 1014 to (-46.98, 290.04, 200) mm, rotated rx -180 ry 0 rz 57.4 deg; joints [53.369, -26.751, 117.303, 53.37, 89.67, 89.557, -1947.405]
  MoveL 1015 to (-42.97, 294.79, 190) mm, rotated rx 180 ry 0 rz 51 deg; joints [53.74, -26.852, 117.772, 53.743, 89.456, 89.258, -1941.005]
  MoveL 1016 to (-38.31, 299.24, 180) mm, rotated rx -180 ry 0 rz 44.31 deg; joints [54.114, -26.948, 118.233, 54.121, 89.247, 88.959, -1934.31]
  MoveL 1017 to (-33.03, 303.26, 170) mm, rotated rx -180 ry 0 rz 37.36 deg; joints [54.492, -27.039, 118.687, 54.503, 89.043, 88.658, -1927.357]
  MoveL 1018 to (-27.19, 306.74, 160) mm, rotated rx -180 ry 0 rz 30.19 deg; joints [54.874, -27.123, 119.133, 54.89, 88.843, 88.355, -1920.187]
  MoveL 1019 to (-20.88, 309.56, 150) mm, rotated rx 180 ry 0 rz 22.84 deg; joints [55.259, -27.199, 119.572, 55.282, 88.648, 88.05, -1912.844]
  MoveL 1020 to (-14.2, 311.65, 140) mm, rotated rx -180 ry 0 rz 15.37 deg; joints [55.647, -27.267, 120.001, 55.678, 88.458, 87.742, -1905.374]
  MoveL 1021 to (-7.28, 312.93, 130) mm, rotated rx -180 ry 0 rz 7.83 deg; joints [56.04, -27.327, 120.422, 56.078, 88.271, 87.432, -1897.828]
  MoveL 1022 to (-0.24, 313.38, 120) mm, rotated rx 180 ry 0 rz 0.26 deg; joints [56.436, -27.377, 120.834, 56.484, 88.09, 87.119, -1890.258]
  MoveL 1023 to (6.77, 312.99, 110) mm, rotated rx -180 ry 0 rz -7.29 deg; joints [56.835, -27.418, 121.236, 56.894, 87.913, 86.803, -1882.715]
  MoveL 1024 to (13.63, 311.79, 100) mm, rotated rx 180 ry 0 rz -14.75 deg; joints [57.239, -27.451, 121.63, 57.308, 87.74, 86.484, -1875.252]
  MoveL 1025 to (20.21, 309.81, 90) mm, rotated rx -180 ry 0 rz -22.08 deg; joints [57.646, -27.474, 122.014, 57.727, 87.572, 86.163, -1867.921]
  MoveL 1026 to (26.38, 307.15, 80) mm, rotated rx -180 ry 0 rz -29.23 deg; joints [58.056, -27.49, 122.39, 58.151, 87.41, 85.839, -1860.769]
  MoveL 1027 to (32.08, 303.89, 70) mm, rotated rx -180 ry 0 rz -36.16 deg; joints [58.471, -27.499, 122.758, 58.579, 87.253, 85.514, -1853.843]
  MoveL 1028 to (37.21, 300.16, 60) mm, rotated rx -180 ry 0 rz -42.82 deg; joints [58.889, -27.502, 123.118, 59.011, 87.101, 85.187, -1847.185]
  MoveL 1029 to (41.73, 296.07, 50) mm, rotated rx -180 ry 0 rz -49.17 deg; joints [59.311, -27.499, 123.471, 59.448, 86.956, 84.859, -1840.833]
  MoveL 1030 to (45.64, 291.75, 40) mm, rotated rx -180 ry 0 rz -55.18 deg; joints [59.736, -27.493, 123.818, 59.888, 86.817, 84.531, -1834.824]
  MoveL 1031 to (48.92, 287.33, 30) mm, rotated rx 180 ry 0 rz -60.81 deg; joints [60.166, -27.483, 124.158, 60.334, 86.685, 84.203, -1829.19]
  MoveL 1032 to (51.6, 282.93, 20) mm, rotated rx -180 ry 0 rz -66.04 deg; joints [60.599, -27.471, 124.492, 60.783, 86.56, 83.876, -1823.962]
  MoveL 1033 to (53.73, 278.68, 10) mm, rotated rx -180 ry 0 rz -70.83 deg; joints [61.035, -27.458, 124.821, 61.236, 86.442, 83.55, -1819.169]
  MoveL 1034 to (55.37, 274.67, 0) mm, rotated rx 180 ry 0 rz -75.16 deg; joints [61.476, -27.444, 125.145, 61.693, 86.331, 83.225, -1814.838]
  MoveL 1035 to (-58.93, 252.99, 290) mm, rotated rx 180 ry 0 rz 96.78 deg; joints [50.189, -25.75, 112.856, 50.225, 91.853, 92.224, -1986.784]
  Set speed (60.0 mm/s)
  MoveL 1036 to (-37.11, 208.63, 290) mm, rotated rx 180 ry 0 rz 144.16 deg; joints [50.189, -25.479, 112.707, 50.222, 91.774, 92.13, -2034.156]
  MoveL 1037 to (55.37, 274.67, 0) mm, rotated rx -180 ry 0 rz -75.16 deg; joints [61.476, -27.444, 125.145, 61.693, 86.331, 83.225, -2174.838]
  Set speed (60.0 mm/s)
  MoveL 1038 to (20.49, 309.71, 0) mm, rotated rx -180 ry 0 rz -22.4 deg; joints [61.476, -27.706, 125.283, 61.686, 86.39, 83.334, -2227.595]
  MoveL 1039 to (55.37, 274.67, 0) mm, rotated rx -180 ry 0 rz -75.16 deg; joints [61.476, -27.444, 125.145, 61.693, 86.331, 83.225, -2174.838]
  Set speed (60.0 mm/s)
  MoveL 1040 to (53.73, 278.68, 10) mm, rotated rx -180 ry 0 rz -70.83 deg; joints [61.035, -27.458, 124.821, 61.236, 86.442, 83.55, -2179.169]
  MoveL 1041 to (51.6, 282.93, 20) mm, rotated rx 180 ry 0 rz -66.04 deg; joints [60.599, -27.471, 124.492, 60.783, 86.56, 83.876, -2183.962]
  MoveL 1042 to (48.92, 287.33, 30) mm, rotated rx -180 ry 0 rz -60.81 deg; joints [60.166, -27.483, 124.158, 60.334, 86.685, 84.203, -2189.19]
  MoveL 1043 to (45.64, 291.75, 40) mm, rotated rx -180 ry 0 rz -55.18 deg; joints [59.736, -27.493, 123.818, 59.888, 86.817, 84.531, -2194.824]
  MoveL 1044 to (41.73, 296.07, 50) mm, rotated rx -180 ry 0 rz -49.17 deg; joints [59.311, -27.499, 123.471, 59.448, 86.956, 84.859, -2200.833]
  MoveL 1045 to (37.21, 300.16, 60) mm, rotated rx -180 ry 0 rz -42.82 deg; joints [58.889, -27.502, 123.118, 59.011, 87.101, 85.187, -2207.185]
  MoveL 1046 to (32.08, 303.89, 70) mm, rotated rx -180 ry 0 rz -36.16 deg; joints [58.471, -27.499, 122.758, 58.579, 87.253, 85.514, -2213.843]
  MoveL 1047 to (26.38, 307.15, 80) mm, rotated rx 180 ry 0 rz -29.23 deg; joints [58.056, -27.49, 122.39, 58.151, 87.41, 85.839, -2220.769]
  MoveL 1048 to (20.21, 309.81, 90) mm, rotated rx -180 ry 0 rz -22.08 deg; joints [57.646, -27.474, 122.014, 57.727, 87.572, 86.163, -2227.921]
  MoveL 1049 to (13.63, 311.79, 100) mm, rotated rx -180 ry 0 rz -14.75 deg; joints [57.239, -27.451, 121.63, 57.308, 87.74, 86.484, -2235.252]
  MoveL 1050 to (6.77, 312.99, 110) mm, rotated rx -180 ry 0 rz -7.29 deg; joints [56.835, -27.418, 121.236, 56.894, 87.913, 86.803, -2242.715]
  MoveL 1051 to (-0.24, 313.38, 120) mm, rotated rx -180 ry 0 rz 0.26 deg; joints [56.436, -27.377, 120.834, 56.484, 88.09, 87.119, -2250.258]
  MoveL 1052 to (-7.28, 312.93, 130) mm, rotated rx -180 ry 0 rz 7.83 deg; joints [56.04, -27.327, 120.422, 56.078, 88.271, 87.432, -2257.828]
  MoveL 1053 to (-14.2, 311.65, 140) mm, rotated rx -180 ry 0 rz 15.37 deg; joints [55.647, -27.267, 120.001, 55.678, 88.458, 87.742, -2265.374]
  MoveL 1054 to (-20.88, 309.56, 150) mm, rotated rx -180 ry 0 rz 22.84 deg; joints [55.259, -27.199, 119.572, 55.282, 88.648, 88.05, -2272.844]
  MoveL 1055 to (-27.19, 306.74, 160) mm, rotated rx 180 ry 0 rz 30.19 deg; joints [54.874, -27.123, 119.133, 54.89, 88.843, 88.355, -2280.187]
  MoveL 1056 to (-33.03, 303.26, 170) mm, rotated rx -180 ry 0 rz 37.36 deg; joints [54.492, -27.039, 118.687, 54.503, 89.043, 88.658, -2287.357]
  MoveL 1057 to (-38.31, 299.24, 180) mm, rotated rx 180 ry 0 rz 44.31 deg; joints [54.114, -26.948, 118.233, 54.121, 89.247, 88.959, -2294.31]
  MoveL 1058 to (-42.97, 294.79, 190) mm, rotated rx -180 ry 0 rz 51 deg; joints [53.74, -26.852, 117.772, 53.743, 89.456, 89.258, -2301.005]
  MoveL 1059 to (-46.98, 290.04, 200) mm, rotated rx -180 ry 0 rz 57.4 deg; joints [53.369, -26.751, 117.303, 53.37, 89.67, 89.557, -2307.405]
  MoveL 1060 to (-50.33, 285.12, 210) mm, rotated rx 180 ry 0 rz 63.48 deg; joints [53.002, -26.646, 116.829, 53.002, 89.89, 89.854, -2313.477]
  MoveL 1061 to (-53.04, 280.16, 220) mm, rotated rx 180 ry 0 rz 69.19 deg; joints [52.638, -26.538, 116.349, 52.638, 90.115, 90.15, -2319.189]
  MoveL 1062 to (-55.14, 275.28, 230) mm, rotated rx 180 ry 0 rz 74.51 deg; joints [52.278, -26.428, 115.864, 52.279, 90.345, 90.446, -2324.512]
  MoveL 1063 to (-56.69, 270.59, 240) mm, rotated rx 180 ry 0 rz 79.42 deg; joints [51.921, -26.316, 115.373, 51.925, 90.582, 90.742, -2329.42]
  MoveL 1064 to (-57.77, 266.19, 250) mm, rotated rx 180 ry 0 rz 83.88 deg; joints [51.568, -26.204, 114.878, 51.575, 90.824, 91.038, -2333.884]
  MoveL 1065 to (-58.44, 262.16, 260) mm, rotated rx -180 ry 0 rz 87.88 deg; joints [51.218, -26.09, 114.379, 51.231, 91.072, 91.334, -2337.879]
  MoveL 1066 to (-58.8, 258.59, 270) mm, rotated rx -180 ry 0 rz 91.38 deg; joints [50.872, -25.977, 113.875, 50.891, 91.326, 91.631, -2341.378]
  MoveL 1067 to (-58.94, 255.51, 280) mm, rotated rx -180 ry 0 rz 94.36 deg; joints [50.529, -25.864, 113.367, 50.555, 91.586, 91.927, -2344.356]
  MoveL 1068 to (-58.93, 252.99, 290) mm, rotated rx 180 ry 0 rz 96.78 deg; joints [50.189, -25.75, 112.856, 50.225, 91.853, 92.224, -2346.784]
  MoveL 1069 to (-37.11, 208.63, 290) mm, rotated rx -180 ry 0 rz 144.16 deg; joints [50.189, -25.479, 112.707, 50.222, 91.774, 92.13, -2394.156]
  Set speed (60.0 mm/s)
  MoveL 1070 to (-39.03, 210.26, 280) mm, rotated rx 180 ry 0 rz 141.88 deg; joints [50.529, -25.585, 113.215, 50.553, 91.506, 91.83, -2391.877]
  MoveL 1071 to (-41.29, 212.35, 270) mm, rotated rx -180 ry 0 rz 139.09 deg; joints [50.872, -25.69, 113.719, 50.888, 91.244, 91.53, -2389.089]
  MoveL 1072 to (-43.78, 214.95, 260) mm, rotated rx -180 ry 0 rz 135.82 deg; joints [51.218, -25.795, 114.218, 51.229, 90.988, 91.23, -2385.82]
  MoveL 1073 to (-46.4, 218.08, 250) mm, rotated rx -180 ry 0 rz 132.1 deg; joints [51.568, -25.9, 114.713, 51.574, 90.738, 90.93, -2382.097]
  MoveL 1074 to (-49.06, 221.75, 240) mm, rotated rx -180 ry 0 rz 127.95 deg; joints [51.921, -26.005, 115.205, 51.924, 90.494, 90.63, -2377.947]
  MoveL 1075 to (-51.62, 225.97, 230) mm, rotated rx -180 ry 0 rz 123.4 deg; joints [52.278, -26.11, 115.692, 52.279, 90.256, 90.331, -2373.396]
  MoveL 1076 to (-53.98, 230.73, 220) mm, rotated rx -180 ry 0 rz 118.47 deg; joints [52.638, -26.216, 116.175, 52.638, 90.025, 90.032, -2368.469]
  MoveL 1077 to (-56, 236.01, 210) mm, rotated rx 180 ry 0 rz 113.19 deg; joints [53.002, -26.322, 116.655, 53.002, 89.8, 89.734, -2363.192]
  MoveL 1078 to (-57.57, 241.75, 200) mm, rotated rx 180 ry 0 rz 107.59 deg; joints [53.369, -26.429, 117.13, 53.371, 89.581, 89.437, -2357.589]
  MoveL 1079 to (-58.59, 247.88, 190) mm, rotated rx -180 ry 0 rz 101.68 deg; joints [53.74, -26.535, 117.602, 53.745, 89.369, 89.14, -2351.684]
  MoveL 1080 to (-58.95, 254.32, 180) mm, rotated rx -180 ry 0 rz 95.5 deg; joints [54.114, -26.641, 118.069, 54.123, 89.163, 88.843, -2345.504]
  MoveL 1081 to (-58.59, 260.95, 170) mm, rotated rx -180 ry 0 rz 89.07 deg; joints [54.492, -26.745, 118.531, 54.505, 88.963, 88.547, -2339.073]
  MoveL 1082 to (-57.45, 267.65, 160) mm, rotated rx -180 ry 0 rz 82.42 deg; joints [54.874, -26.848, 118.987, 54.892, 88.769, 88.25, -2332.419]
  MoveL 1083 to (-55.51, 274.28, 150) mm, rotated rx -180 ry 0 rz 75.57 deg; joints [55.259, -26.948, 119.438, 55.284, 88.581, 87.953, -2325.573]
  MoveL 1084 to (-52.77, 280.72, 140) mm, rotated rx -180 ry 0 rz 68.57 deg; joints [55.647, -27.045, 119.883, 55.68, 88.399, 87.656, -2318.565]
  MoveL 1085 to (-49.26, 286.82, 130) mm, rotated rx -180 ry 0 rz 61.43 deg; joints [56.04, -27.137, 120.322, 56.081, 88.222, 87.358, -2311.431]
  MoveL 1086 to (-45.04, 292.47, 120) mm, rotated rx -180 ry 0 rz 54.21 deg; joints [56.436, -27.224, 120.753, 56.486, 88.05, 87.058, -2304.209]
  MoveL 1087 to (-40.19, 297.56, 110) mm, rotated rx -180 ry 0 rz 46.94 deg; joints [56.835, -27.304, 121.176, 56.895, 87.883, 86.758, -2296.94]
  MoveL 1088 to (-34.83, 302, 100) mm, rotated rx 180 ry 0 rz 39.67 deg; joints [57.239, -27.378, 121.591, 57.309, 87.721, 86.455, -2289.668]
  MoveL 1089 to (-29.06, 305.72, 90) mm, rotated rx -180 ry 0 rz 32.44 deg; joints [57.646, -27.444, 121.998, 57.728, 87.565, 86.15, -2282.441]
  MoveL 1090 to (-23.03, 308.7, 80) mm, rotated rx -180 ry 0 rz 25.31 deg; joints [58.056, -27.502, 122.396, 58.15, 87.413, 85.844, -2275.308]
  MoveL 1091 to (-16.86, 310.92, 70) mm, rotated rx 180 ry 0 rz 18.32 deg; joints [58.471, -27.552, 122.786, 58.577, 87.266, 85.535, -2268.32]
  MoveL 1092 to (-10.69, 312.41, 60) mm, rotated rx -180 ry 0 rz 11.53 deg; joints [58.889, -27.594, 123.167, 59.009, 87.124, 85.224, -2261.529]
  MoveL 1093 to (-4.64, 313.2, 50) mm, rotated rx 180 ry 0 rz 4.98 deg; joints [59.311, -27.628, 123.539, 59.445, 86.987, 84.912, -2254.983]
  MoveL 1094 to (1.18, 313.37, 40) mm, rotated rx -180 ry 0 rz -1.27 deg; joints [59.736, -27.655, 123.903, 59.885, 86.856, 84.598, -2248.733]
  MoveL 1095 to (6.67, 313.01, 30) mm, rotated rx -180 ry 0 rz -7.17 deg; joints [60.166, -27.676, 124.259, 60.329, 86.73, 84.283, -2242.826]
  MoveL 1096 to (11.76, 312.2, 20) mm, rotated rx -180 ry 0 rz -12.69 deg; joints [60.599, -27.69, 124.608, 60.777, 86.61, 83.967, -2237.306]
  MoveL 1097 to (16.38, 311.06, 10) mm, rotated rx -180 ry 0 rz -17.78 deg; joints [61.035, -27.7, 124.949, 61.23, 86.497, 83.65, -2232.216]
  MoveL 1098 to (20.49, 309.71, 0) mm, rotated rx -180 ry 0 rz -22.4 deg; joints [61.476, -27.706, 125.283, 61.686, 86.39, 83.334, -2227.595]
  MoveL 1099 to (-37.11, 208.63, 290) mm, rotated rx -180 ry 0 rz 144.16 deg; joints [50.189, -25.479, 112.707, 50.222, 91.774, 92.13, -2394.156]
  Set speed (60.0 mm/s)
  MoveL 1100 to (-43.85, 188.95, 290) mm, rotated rx -180 ry 0 rz 148.32 deg; joints [50.189, -24.124, 111.947, 50.209, 91.394, 91.673, -2398.321]
  MoveL 1101 to (20.49, 309.71, 0) mm, rotated rx -180 ry 0 rz -22.4 deg; joints [61.476, -27.706, 125.283, 61.686, 86.39, 83.334, -2227.595]
  Set speed (60.0 mm/s)
  MoveL 1102 to (20.57, 330.51, 0) mm, rotated rx -180 ry 0 rz -16.27 deg; joints [61.476, -26.245, 124.499, 61.726, 86.069, 82.736, -2233.733]
  MoveL 1103 to (20.49, 309.71, 0) mm, rotated rx -180 ry 0 rz -22.4 deg; joints [61.476, -27.706, 125.283, 61.686, 86.39, 83.334, -2227.595]
  Set speed (60.0 mm/s)
  MoveL 1104 to (16.38, 311.06, 10) mm, rotated rx -180 ry 0 rz -17.78 deg; joints [61.035, -27.7, 124.949, 61.23, 86.497, 83.65, -2232.216]
  MoveL 1105 to (11.76, 312.2, 20) mm, rotated rx -180 ry 0 rz -12.69 deg; joints [60.599, -27.69, 124.608, 60.777, 86.61, 83.967, -2237.306]
  MoveL 1106 to (6.67, 313.01, 30) mm, rotated rx -180 ry 0 rz -7.17 deg; joints [60.166, -27.676, 124.259, 60.329, 86.73, 84.283, -2242.826]
  MoveL 1107 to (1.18, 313.37, 40) mm, rotated rx -180 ry 0 rz -1.27 deg; joints [59.736, -27.655, 123.903, 59.885, 86.856, 84.598, -2248.733]
  MoveL 1108 to (-4.64, 313.2, 50) mm, rotated rx 180 ry 0 rz 4.98 deg; joints [59.311, -27.628, 123.539, 59.445, 86.987, 84.912, -2254.983]
  MoveL 1109 to (-10.69, 312.41, 60) mm, rotated rx -180 ry 0 rz 11.53 deg; joints [58.889, -27.594, 123.167, 59.009, 87.124, 85.224, -2261.529]
  MoveL 1110 to (-16.86, 310.92, 70) mm, rotated rx 180 ry 0 rz 18.32 deg; joints [58.471, -27.552, 122.786, 58.577, 87.266, 85.535, -2268.32]
  MoveL 1111 to (-23.03, 308.7, 80) mm, rotated rx -180 ry 0 rz 25.31 deg; joints [58.056, -27.502, 122.396, 58.15, 87.413, 85.844, -2275.308]
  MoveL 1112 to (-29.06, 305.72, 90) mm, rotated rx -180 ry 0 rz 32.44 deg; joints [57.646, -27.444, 121.998, 57.728, 87.565, 86.15, -2282.441]
  MoveL 1113 to (-34.83, 302, 100) mm, rotated rx -180 ry 0 rz 39.67 deg; joints [57.239, -27.378, 121.591, 57.309, 87.721, 86.455, -2289.668]
  MoveL 1114 to (-40.19, 297.56, 110) mm, rotated rx -180 ry 0 rz 46.94 deg; joints [56.835, -27.304, 121.176, 56.895, 87.883, 86.758, -2296.94]
  MoveL 1115 to (-45.04, 292.47, 120) mm, rotated rx -180 ry 0 rz 54.21 deg; joints [56.436, -27.224, 120.753, 56.486, 88.05, 87.058, -2304.209]
  MoveL 1116 to (-49.26, 286.82, 130) mm, rotated rx -180 ry 0 rz 61.43 deg; joints [56.04, -27.137, 120.322, 56.081, 88.222, 87.358, -2311.431]
  MoveL 1117 to (-52.77, 280.72, 140) mm, rotated rx -180 ry 0 rz 68.57 deg; joints [55.647, -27.045, 119.883, 55.68, 88.399, 87.656, -2318.565]
  MoveL 1118 to (-55.51, 274.28, 150) mm, rotated rx 180 ry 0 rz 75.57 deg; joints [55.259, -26.948, 119.438, 55.284, 88.581, 87.953, -2325.573]
  MoveL 1119 to (-57.45, 267.65, 160) mm, rotated rx 180 ry 0 rz 82.42 deg; joints [54.874, -26.848, 118.987, 54.892, 88.769, 88.25, -2332.419]
  MoveL 1120 to (-58.59, 260.95, 170) mm, rotated rx -180 ry 0 rz 89.07 deg; joints [54.492, -26.745, 118.531, 54.505, 88.963, 88.547, -2339.073]
  MoveL 1121 to (-58.95, 254.32, 180) mm, rotated rx 180 ry 0 rz 95.5 deg; joints [54.114, -26.641, 118.069, 54.123, 89.163, 88.843, -2345.504]
  MoveL 1122 to (-58.59, 247.88, 190) mm, rotated rx 180 ry 0 rz 101.68 deg; joints [53.74, -26.535, 117.602, 53.745, 89.369, 89.14, -2351.684]
  MoveL 1123 to (-57.57, 241.75, 200) mm, rotated rx -180 ry 0 rz 107.59 deg; joints [53.369, -26.429, 117.13, 53.371, 89.581, 89.437, -2357.589]
  MoveL 1124 to (-56, 236.01, 210) mm, rotated rx -180 ry 0 rz 113.19 deg; joints [53.002, -26.322, 116.655, 53.002, 89.8, 89.734, -2363.192]
  MoveL 1125 to (-53.98, 230.73, 220) mm, rotated rx -180 ry 0 rz 118.47 deg; joints [52.638, -26.216, 116.175, 52.638, 90.025, 90.032, -2368.469]
  MoveL 1126 to (-51.62, 225.97, 230) mm, rotated rx -180 ry 0 rz 123.4 deg; joints [52.278, -26.11, 115.692, 52.279, 90.256, 90.331, -2373.396]
  MoveL 1127 to (-49.06, 221.75, 240) mm, rotated rx -180 ry 0 rz 127.95 deg; joints [51.921, -26.005, 115.205, 51.924, 90.494, 90.63, -2377.947]
  MoveL 1128 to (-46.4, 218.08, 250) mm, rotated rx -180 ry 0 rz 132.1 deg; joints [51.568, -25.9, 114.713, 51.574, 90.738, 90.93, -2382.097]
  MoveL 1129 to (-43.78, 214.95, 260) mm, rotated rx -180 ry 0 rz 135.82 deg; joints [51.218, -25.795, 114.218, 51.229, 90.988, 91.23, -2385.82]
  MoveL 1130 to (-41.29, 212.35, 270) mm, rotated rx -180 ry 0 rz 139.09 deg; joints [50.872, -25.69, 113.719, 50.888, 91.244, 91.53, -2389.089]
  MoveL 1131 to (-39.03, 210.26, 280) mm, rotated rx -180 ry 0 rz 141.88 deg; joints [50.529, -25.585, 113.215, 50.553, 91.506, 91.83, -2391.877]
  MoveL 1132 to (-37.11, 208.63, 290) mm, rotated rx -180 ry 0 rz 144.16 deg; joints [50.189, -25.479, 112.707, 50.222, 91.774, 92.13, -2394.156]
  MoveL 1133 to (-43.85, 188.95, 290) mm, rotated rx 180 ry 0 rz 148.32 deg; joints [50.189, -24.124, 111.947, 50.209, 91.394, 91.673, -2398.321]
  Set speed (60.0 mm/s)
  MoveL 1134 to (-46.6, 190.89, 280) mm, rotated rx 180 ry 0 rz 146.01 deg; joints [50.529, -24.224, 112.453, 50.542, 91.126, 91.368, -2396.008]
  MoveL 1135 to (-49.86, 193.4, 270) mm, rotated rx -180 ry 0 rz 143.18 deg; joints [50.872, -24.324, 112.955, 50.88, 90.864, 91.062, -2393.179]
  MoveL 1136 to (-53.49, 196.56, 260) mm, rotated rx 180 ry 0 rz 139.86 deg; joints [51.218, -24.423, 113.452, 51.222, 90.608, 90.757, -2389.865]
  MoveL 1137 to (-57.36, 200.4, 250) mm, rotated rx -180 ry 0 rz 136.1 deg; joints [51.568, -24.521, 113.945, 51.569, 90.358, 90.451, -2386.095]
  MoveL 1138 to (-61.34, 204.96, 240) mm, rotated rx -180 ry 0 rz 131.9 deg; joints [51.921, -24.62, 114.435, 51.921, 90.115, 90.146, -2381.899]
  MoveL 1139 to (-65.27, 210.27, 230) mm, rotated rx -180 ry 0 rz 127.3 deg; joints [52.278, -24.719, 114.92, 52.278, 89.877, 89.841, -2377.303]
  MoveL 1140 to (-68.98, 216.33, 220) mm, rotated rx -180 ry 0 rz 122.34 deg; joints [52.638, -24.819, 115.402, 52.64, 89.646, 89.537, -2372.338]
  MoveL 1141 to (-72.31, 223.11, 210) mm, rotated rx -180 ry 0 rz 117.03 deg; joints [53.002, -24.919, 115.879, 53.006, 89.422, 89.233, -2367.029]
  MoveL 1142 to (-75.1, 230.56, 200) mm, rotated rx -180 ry 0 rz 111.4 deg; joints [53.369, -25.019, 116.353, 53.377, 89.204, 88.929, -2361.404]
  MoveL 1143 to (-77.2, 238.6, 190) mm, rotated rx -180 ry 0 rz 105.49 deg; joints [53.74, -25.12, 116.823, 53.752, 88.993, 88.626, -2355.49]
  MoveL 1144 to (-78.47, 247.13, 180) mm, rotated rx -180 ry 0 rz 99.32 deg; joints [54.114, -25.22, 117.289, 54.132, 88.788, 88.324, -2349.316]
  MoveL 1145 to (-78.79, 256, 170) mm, rotated rx -180 ry 0 rz 92.91 deg; joints [54.492, -25.32, 117.75, 54.517, 88.589, 88.021, -2342.909]
  MoveL 1146 to (-78.09, 265.05, 160) mm, rotated rx -180 ry 0 rz 86.3 deg; joints [54.874, -25.418, 118.206, 54.906, 88.396, 87.719, -2336.299]
  MoveL 1147 to (-76.31, 274.12, 150) mm, rotated rx -180 ry 0 rz 79.52 deg; joints [55.259, -25.513, 118.656, 55.299, 88.21, 87.417, -2329.517]
  MoveL 1148 to (-73.44, 283.02, 140) mm, rotated rx -180 ry 0 rz 72.6 deg; joints [55.647, -25.606, 119.1, 55.697, 88.029, 87.114, -2322.596]
  MoveL 1149 to (-69.5, 291.57, 130) mm, rotated rx -180 ry 0 rz 65.57 deg; joints [56.04, -25.694, 119.538, 56.099, 87.854, 86.81, -2315.57]
  MoveL 1150 to (-64.57, 299.61, 120) mm, rotated rx 180 ry 0 rz 58.48 deg; joints [56.436, -25.778, 119.969, 56.506, 87.684, 86.506, -2308.477]
  MoveL 1151 to (-58.74, 306.97, 110) mm, rotated rx -180 ry 0 rz 51.35 deg; joints [56.835, -25.856, 120.392, 56.918, 87.52, 86.2, -2301.355]
  MoveL 1152 to (-52.14, 313.53, 100) mm, rotated rx -180 ry 0 rz 44.25 deg; joints [57.239, -25.927, 120.808, 57.333, 87.361, 85.893, -2294.246]
  MoveL 1153 to (-44.91, 319.19, 90) mm, rotated rx -180 ry 0 rz 37.19 deg; joints [57.646, -25.991, 121.215, 57.753, 87.207, 85.584, -2287.194]
  MoveL 1154 to (-37.24, 323.88, 80) mm, rotated rx 180 ry 0 rz 30.24 deg; joints [58.056, -26.048, 121.613, 58.178, 87.059, 85.273, -2280.242]
  MoveL 1155 to (-29.3, 327.59, 70) mm, rotated rx -180 ry 0 rz 23.44 deg; joints [58.471, -26.097, 122.003, 58.607, 86.915, 84.961, -2273.438]
  MoveL 1156 to (-21.27, 330.31, 60) mm, rotated rx 180 ry 0 rz 16.83 deg; joints [58.889, -26.138, 122.384, 59.04, 86.777, 84.646, -2266.828]
  MoveL 1157 to (-13.31, 332.11, 50) mm, rotated rx 180 ry 0 rz 10.46 deg; joints [59.311, -26.171, 122.757, 59.477, 86.644, 84.33, -2260.456]
  MoveL 1158 to (-5.58, 333.04, 40) mm, rotated rx -180 ry 0 rz 4.37 deg; joints [59.736, -26.197, 123.121, 59.919, 86.517, 84.013, -2254.37]
  MoveL 1159 to (1.77, 333.22, 30) mm, rotated rx -180 ry 0 rz -1.39 deg; joints [60.166, -26.217, 123.476, 60.364, 86.396, 83.695, -2248.612]
  MoveL 1160 to (8.64, 332.76, 20) mm, rotated rx -180 ry 0 rz -6.77 deg; joints [60.599, -26.231, 123.825, 60.814, 86.281, 83.375, -2243.227]
  MoveL 1161 to (14.93, 331.81, 10) mm, rotated rx -180 ry 0 rz -11.75 deg; joints [61.035, -26.24, 124.165, 61.268, 86.172, 83.056, -2238.254]
  MoveL 1162 to (20.57, 330.51, 0) mm, rotated rx 180 ry 0 rz -16.27 deg; joints [61.476, -26.245, 124.499, 61.726, 86.069, 82.736, -2233.733]
  MoveL 1163 to (-43.85, 188.95, 290) mm, rotated rx 180 ry 0 rz 148.32 deg; joints [50.189, -24.124, 111.947, 50.209, 91.394, 91.673, -2398.321]
  Set speed (60.0 mm/s)
  MoveL 1164 to (-28.22, 202.67, 290) mm, rotated rx 180 ry 0 rz 153.79 deg; joints [50.189, -25.444, 112.688, 50.221, 91.764, 92.118, -2403.793]
  MoveL 1165 to (20.57, 330.51, 0) mm, rotated rx -180 ry 0 rz -16.27 deg; joints [61.476, -26.245, 124.499, 61.726, 86.069, 82.736, -2233.733]
  Set speed (60.0 mm/s)
  MoveL 1166 to (10.16, 312.5, 0) mm, rotated rx 180 ry 0 rz -10.95 deg; joints [61.476, -27.728, 125.294, 61.686, 86.395, 83.343, -2239.047]
  MoveL 1167 to (20.57, 330.51, 0) mm, rotated rx 180 ry 0 rz -16.27 deg; joints [61.476, -26.245, 124.499, 61.726, 86.069, 82.736, -2233.733]
  Set speed (60.0 mm/s)
  MoveL 1168 to (14.93, 331.81, 10) mm, rotated rx -180 ry 0 rz -11.75 deg; joints [61.035, -26.24, 124.165, 61.268, 86.172, 83.056, -2238.254]
  MoveL 1169 to (8.64, 332.76, 20) mm, rotated rx -180 ry 0 rz -6.77 deg; joints [60.599, -26.231, 123.825, 60.814, 86.281, 83.375, -2243.227]
  MoveL 1170 to (1.77, 333.22, 30) mm, rotated rx -180 ry 0 rz -1.39 deg; joints [60.166, -26.217, 123.476, 60.364, 86.396, 83.695, -2248.612]
  MoveL 1171 to (-5.58, 333.04, 40) mm, rotated rx -180 ry 0 rz 4.37 deg; joints [59.736, -26.197, 123.121, 59.919, 86.517, 84.013, -2254.37]
  MoveL 1172 to (-13.31, 332.11, 50) mm, rotated rx 180 ry 0 rz 10.46 deg; joints [59.311, -26.171, 122.757, 59.477, 86.644, 84.33, -2260.456]
  MoveL 1173 to (-21.27, 330.31, 60) mm, rotated rx 180 ry 0 rz 16.83 deg; joints [58.889, -26.138, 122.384, 59.04, 86.777, 84.646, -2266.828]
  MoveL 1174 to (-29.3, 327.59, 70) mm, rotated rx -180 ry 0 rz 23.44 deg; joints [58.471, -26.097, 122.003, 58.607, 86.915, 84.961, -2273.438]
  MoveL 1175 to (-37.24, 323.88, 80) mm, rotated rx 180 ry 0 rz 30.24 deg; joints [58.056, -26.048, 121.613, 58.178, 87.059, 85.273, -2280.242]
  MoveL 1176 to (-44.91, 319.19, 90) mm, rotated rx -180 ry 0 rz 37.19 deg; joints [57.646, -25.991, 121.215, 57.753, 87.207, 85.584, -2287.194]
  MoveL 1177 to (-52.14, 313.53, 100) mm, rotated rx -180 ry 0 rz 44.25 deg; joints [57.239, -25.927, 120.808, 57.333, 87.361, 85.893, -2294.246]
  MoveL 1178 to (-58.74, 306.97, 110) mm, rotated rx -180 ry 0 rz 51.35 deg; joints [56.835, -25.856, 120.392, 56.918, 87.52, 86.2, -2301.355]
  MoveL 1179 to (-64.57, 299.61, 120) mm, rotated rx 180 ry 0 rz 58.48 deg; joints [56.436, -25.778, 119.969, 56.506, 87.684, 86.506, -2308.477]
  MoveL 1180 to (-69.5, 291.57, 130) mm, rotated rx -180 ry 0 rz 65.57 deg; joints [56.04, -25.694, 119.538, 56.099, 87.854, 86.81, -2315.57]
  MoveL 1181 to (-73.44, 283.02, 140) mm, rotated rx -180 ry 0 rz 72.6 deg; joints [55.647, -25.606, 119.1, 55.697, 88.029, 87.114, -2322.596]
  MoveL 1182 to (-76.31, 274.12, 150) mm, rotated rx -180 ry 0 rz 79.52 deg; joints [55.259, -25.513, 118.656, 55.299, 88.21, 87.417, -2329.517]
  MoveL 1183 to (-78.09, 265.05, 160) mm, rotated rx -180 ry 0 rz 86.3 deg; joints [54.874, -25.418, 118.206, 54.906, 88.396, 87.719, -2336.299]
  MoveL 1184 to (-78.79, 256, 170) mm, rotated rx -180 ry 0 rz 92.91 deg; joints [54.492, -25.32, 117.75, 54.517, 88.589, 88.021, -2342.909]
  MoveL 1185 to (-78.47, 247.13, 180) mm, rotated rx -180 ry 0 rz 99.32 deg; joints [54.114, -25.22, 117.289, 54.132, 88.788, 88.324, -2349.316]
  MoveL 1186 to (-77.2, 238.6, 190) mm, rotated rx -180 ry 0 rz 105.49 deg; joints [53.74, -25.12, 116.823, 53.752, 88.993, 88.626, -2355.49]
  MoveL 1187 to (-75.1, 230.56, 200) mm, rotated rx -180 ry 0 rz 111.4 deg; joints [53.369, -25.019, 116.353, 53.377, 89.204, 88.929, -2361.404]
  MoveL 1188 to (-72.31, 223.11, 210) mm, rotated rx -180 ry 0 rz 117.03 deg; joints [53.002, -24.919, 115.879, 53.006, 89.422, 89.233, -2367.029]
  MoveL 1189 to (-68.98, 216.33, 220) mm, rotated rx -180 ry 0 rz 122.34 deg; joints [52.638, -24.819, 115.402, 52.64, 89.646, 89.537, -2372.338]
  MoveL 1190 to (-65.27, 210.27, 230) mm, rotated rx -180 ry 0 rz 127.3 deg; joints [52.278, -24.719, 114.92, 52.278, 89.877, 89.841, -2377.303]
  MoveL 1191 to (-61.34, 204.96, 240) mm, rotated rx -180 ry 0 rz 131.9 deg; joints [51.921, -24.62, 114.435, 51.921, 90.115, 90.146, -2381.899]
  MoveL 1192 to (-57.36, 200.4, 250) mm, rotated rx -180 ry 0 rz 136.1 deg; joints [51.568, -24.521, 113.945, 51.569, 90.358, 90.451, -2386.095]
  MoveL 1193 to (-53.49, 196.56, 260) mm, rotated rx 180 ry 0 rz 139.86 deg; joints [51.218, -24.423, 113.452, 51.222, 90.608, 90.757, -2389.865]
  MoveL 1194 to (-49.86, 193.4, 270) mm, rotated rx -180 ry 0 rz 143.18 deg; joints [50.872, -24.324, 112.955, 50.88, 90.864, 91.062, -2393.179]
  MoveL 1195 to (-46.6, 190.89, 280) mm, rotated rx 180 ry 0 rz 146.01 deg; joints [50.529, -24.224, 112.453, 50.542, 91.126, 91.368, -2396.008]
  MoveL 1196 to (-43.85, 188.95, 290) mm, rotated rx 180 ry 0 rz 148.32 deg; joints [50.189, -24.124, 111.947, 50.209, 91.394, 91.673, -2398.321]
  MoveL 1197 to (-28.22, 202.67, 290) mm, rotated rx -180 ry 0 rz 153.79 deg; joints [50.189, -25.444, 112.688, 50.221, 91.764, 92.118, -2403.793]
  Set speed (60.0 mm/s)
  MoveL 1198 to (-30.4, 203.93, 280) mm, rotated rx -180 ry 0 rz 151.53 deg; joints [50.529, -25.548, 113.195, 50.552, 91.495, 91.817, -2401.533]
  MoveL 1199 to (-33, 205.58, 270) mm, rotated rx -180 ry 0 rz 148.77 deg; joints [50.872, -25.65, 113.697, 50.888, 91.232, 91.515, -2398.768]
  MoveL 1200 to (-35.92, 207.69, 260) mm, rotated rx -180 ry 0 rz 145.53 deg; joints [51.218, -25.752, 114.194, 51.228, 90.975, 91.214, -2395.528]
  MoveL 1201 to (-39.07, 210.28, 250) mm, rotated rx -180 ry 0 rz 141.84 deg; joints [51.568, -25.853, 114.688, 51.574, 90.724, 90.913, -2391.841]
  MoveL 1202 to (-42.34, 213.41, 240) mm, rotated rx 180 ry 0 rz 137.73 deg; joints [51.921, -25.954, 115.177, 51.924, 90.479, 90.612, -2387.735]
  MoveL 1203 to (-45.62, 217.1, 230) mm, rotated rx -180 ry 0 rz 133.24 deg; joints [52.278, -26.056, 115.662, 52.279, 90.241, 90.311, -2383.236]
  MoveL 1204 to (-48.8, 221.36, 220) mm, rotated rx -180 ry 0 rz 128.37 deg; joints [52.638, -26.158, 116.144, 52.638, 90.009, 90.011, -2378.371]
  MoveL 1205 to (-51.74, 226.19, 210) mm, rotated rx 180 ry 0 rz 123.16 deg; joints [53.002, -26.261, 116.622, 53.003, 89.783, 89.712, -2373.164]
  MoveL 1206 to (-54.33, 231.55, 200) mm, rotated rx -180 ry 0 rz 117.64 deg; joints [53.369, -26.364, 117.095, 53.371, 89.563, 89.413, -2367.64]
  MoveL 1207 to (-56.44, 237.4, 190) mm, rotated rx -180 ry 0 rz 111.82 deg; joints [53.74, -26.467, 117.565, 53.745, 89.351, 89.115, -2361.825]
  MoveL 1208 to (-57.96, 243.66, 180) mm, rotated rx -180 ry 0 rz 105.74 deg; joints [54.114, -26.571, 118.031, 54.123, 89.144, 88.817, -2355.742]
  MoveL 1209 to (-58.8, 250.25, 170) mm, rotated rx 180 ry 0 rz 99.42 deg; joints [54.492, -26.674, 118.493, 54.506, 88.944, 88.52, -2349.418]
  MoveL 1210 to (-58.89, 257.04, 160) mm, rotated rx -180 ry 0 rz 92.88 deg; joints [54.874, -26.777, 118.949, 54.893, 88.75, 88.223, -2342.877]
  MoveL 1211 to (-58.18, 263.92, 150) mm, rotated rx -180 ry 0 rz 86.15 deg; joints [55.259, -26.878, 119.401, 55.285, 88.562, 87.926, -2336.149]
  MoveL 1212 to (-56.65, 270.74, 140) mm, rotated rx -180 ry 0 rz 79.26 deg; joints [55.647, -26.976, 119.847, 55.681, 88.381, 87.629, -2329.263]
  MoveL 1213 to (-54.3, 277.38, 130) mm, rotated rx -180 ry 0 rz 72.25 deg; joints [56.04, -27.071, 120.286, 56.082, 88.204, 87.332, -2322.251]
  MoveL 1214 to (-51.17, 283.7, 120) mm, rotated rx 180 ry 0 rz 65.15 deg; joints [56.436, -27.161, 120.719, 56.487, 88.034, 87.034, -2315.149]
  MoveL 1215 to (-47.33, 289.58, 110) mm, rotated rx -180 ry 0 rz 57.99 deg; joints [56.835, -27.247, 121.145, 56.896, 87.868, 86.735, -2307.994]
  MoveL 1216 to (-42.85, 294.92, 100) mm, rotated rx -180 ry 0 rz 50.83 deg; joints [57.239, -27.326, 121.564, 57.31, 87.708, 86.434, -2300.828]
  MoveL 1217 to (-37.86, 299.62, 90) mm, rotated rx -180 ry 0 rz 43.7 deg; joints [57.646, -27.399, 121.974, 57.728, 87.553, 86.132, -2293.695]
  MoveL 1218 to (-32.46, 303.64, 80) mm, rotated rx -180 ry 0 rz 36.64 deg; joints [58.056, -27.464, 122.377, 58.151, 87.403, 85.829, -2286.643]
  MoveL 1219 to (-26.8, 306.94, 70) mm, rotated rx -180 ry 0 rz 29.72 deg; joints [58.471, -27.522, 122.77, 58.578, 87.258, 85.523, -2279.72]
  MoveL 1220 to (-21, 309.52, 60) mm, rotated rx 180 ry 0 rz 22.98 deg; joints [58.889, -27.572, 123.155, 59.009, 87.118, 85.216, -2272.977]
  MoveL 1221 to (-15.19, 311.39, 50) mm, rotated rx 180 ry 0 rz 16.46 deg; joints [59.311, -27.614, 123.532, 59.445, 86.984, 84.906, -2266.464]
  MoveL 1222 to (-9.5, 312.61, 40) mm, rotated rx -180 ry 0 rz 10.23 deg; joints [59.736, -27.649, 123.9, 59.885, 86.854, 84.595, -2260.231]
  MoveL 1223 to (-4.03, 313.25, 30) mm, rotated rx 180 ry 0 rz 4.33 deg; joints [60.166, -27.677, 124.26, 60.329, 86.731, 84.283, -2254.327]
  MoveL 1224 to (1.12, 313.37, 20) mm, rotated rx -180 ry 0 rz -1.2 deg; joints [60.599, -27.699, 124.612, 60.777, 86.612, 83.97, -2248.799]
  MoveL 1225 to (5.87, 313.09, 10) mm, rotated rx 180 ry 0 rz -6.31 deg; joints [61.035, -27.716, 124.957, 61.229, 86.5, 83.657, -2243.692]
  MoveL 1226 to (10.16, 312.5, 0) mm, rotated rx -180 ry 0 rz -10.95 deg; joints [61.476, -27.728, 125.294, 61.686, 86.395, 83.343, -2239.047]
  Set speed (1000.0 mm/s)
  MoveL 1227 to (10.16, 312.5, 0) mm, rotated rx -180 ry 0 rz -10.95 deg; joints [61.476, -27.728, 125.294, 61.686, 86.395, 83.343, -2239.047]
